(*####################### Folgende Werte sind Regelparameter und müssen initialisiert werden##########################*)
	T_ZYKL: REAL:=0.001;(*Zykluszeit in s, in der dieser Baustein aufgerufen wird*)
	C_INVERS:BOOL:=FALSE; (*Zählrichtungsumkehr*)
	IBW:LREAL:=0.1; (*Istbewertung in mm pro Increment*)
	REFVEL1:REAL:=10; (*Referenzfahrtgeschwindigkeit, um Endschalter zu suchen, positive oder negative Werte:1=langsam,2=schnell*)
	REFVEL2:REAL:=-10; (*Referenzfahrtgeschwindigkeit, um vom Endschalter weg die Nullspur zu suchen,  positive oder negative Werte:1=langsam,2=schnel*)
	REF_ON:BOOL; (*Referenzfahrt ohne Nullspur, d.h. bei negtiver Flanke des Endsch. wird Istwert gesetzt*)
	OPTI_KURZ:BOOL;(*optimierung bei kurzer Strecke:Ist der Verfahrweg kleiner als 2*S_SCHLEICH, dann wird auf halbem Weg beschleunugt(EIL) und auf halbem abgebremst (SCHLEICH*)
	WAITTIME_INV:REAL:=0.3;(*Wartezeit bei Richtungsumkehr in SEC*)
	WAIT_Restart_akt:BOOL;(* Wartezeit bei wiederStarten aktiv: wenn der Antrieb abgeschaltet wird, dann bleiben die Ausgänge MINDESTENS "Waittime_INV" abgeschaltet (notwendig bei 24V-DC Lineramotoren) *)
	S_SCHLEICH: REAL;(*Schleichweg*)
	S_STOP: REAL;(*Vorabschaltdifferenz, innerhalb diesem Fenster wird nicht positioniert, sondern PEH ausgegeben!*)
	T_VERZ_STILL:REAL;(*Verzögerungszeit zum Ansprechen der Stillstandsüberwachung, Sekunden*)
	IstWertOffset:LREAL;(*Offset, der  auf den Istwert(Benutzereinheit bzw. mm) Online aufgerechnent wird*)
	MaxIstDiff_pro_Zykl: REAL;(*Einheit: Benutzer (mm) . Wenn zwischen 2 Zyklen eine Istwertänderung (Benutzereinheit bzw. mm) von mehr als dieser Wert auftritt, wird SYNC gelöscht*)
	Loop_val: REAL;		(*schleife fahren: 0=nein; ansonsten: Es wird um den Betrag von S_STOP+Loop_Val vom Ziel weggefahren, abhängig vom Vorzeiche: + in pos.
							Richtung,- in neg. Richtung). Loop_val wird nur bei pos. Flanke Start oder Änderung der Sollpos bei aktivem Start ausgewertet, d.h. eine Änderung während dem Positionieren wird ignoriert*)
END_VAR
VAR_OUTPUT
	DAT_TO_PLC:TES_Achse_IN;(*Übergabe der Parameter zum Anwenderprogramm *)
	COUNT_CTRL: BYTE;(*Verknüpfung mit COUNTER CTRL*)
	EIL_OUT:BOOL;(*Verknüpfung mit Ausgang schnell*)
	VOR_OUT:BOOL;(*Verknüpfung mit Ausgang vor*)
	ZUR_OUT:BOOL;(*Verknüpfung mit Ausgang zur*)
	ERR_INIT:BOOL:=TRUE;(*Fehler bei initialisierung oder noch nicht initialisiert*)
END_VAR

VAR

(*########################################Ausgangsvariabeln vom Baustein -> STRUKTUR(IN) ###################################*)
	IstPos: LREAL;(*Istposition Achse *)
	SYNC: BOOL := FALSE;
	PEH:BOOL;

(*####################################Folgende Daten werden intern berechnet und verwendet#####################################*)
	OFFSET_INC: LREAL;
	COUNT_INC: DWORD;(*Zähler-INCREMENTE*)
	COUNT_INC_LAST: DWORD;(*Zähler-INCREMENTE des letzten Zyklus, sofern Zähler-Val gültig war*)
	REFSTATUS: INT; (*0=aus,1=suche Endsch;2=Suche neg.Flanke Endsch;3=suche Nullspur,...7=beendet*)
	LAST_COUNT_CTRL: BYTE;
	V_SOLL:REAL;(*Sollgeschwindifkeit, die aufgrund der berechnungen resultiert.V_F_T wird durch V_Soll UND den zulässigen Rampen (zulässige Geschw.-Änderung pro Zyklus) berechnet*)
	Zieldiff_Pos: LREAL;(*POS-Modus: Differenz zum Ziel*)
	Start_Pos_LAST: BOOL;
	SollPos: LREAL;(*Zielposition bei Positionierung*)
	MODULOVAL_INC:REAL;(*Wert in Incrementen für MODULO-Funktion*)
	TIME_VOR: REAL;
	TIME_ZUR: REAL;
	MODULO_ERG: LREAL;
	StartFRG_Pos: BOOL;
	S_SCHLEICH_I: REAL;(*Schleichweg, Intern. Der Wert S_SCHLEICH (VAR_INPUT) wird auf S_SCHLEICH_I kopiert, außer bei optimierung für kurze Strecken *)
	T_STILLST: REAL;(* abgelaufene Stillstandszeit*)
	SetIstPos: BOOL;
	IstPos_LAST: LREAL;
	IstWertOffset_LAST: LREAL;
	Loop_akt: BOOL;(*Schleife-fahren ist aktiv*)
	c_Loop_val: REAL;(* Kopie von LoopVAL*)
	EncBitMask: DWORD;
	CountLimit1: DWORD;
	CountLimit2: DWORD;
	EmptyBits: INT;
END_VAR

SetIstPos:=FALSE;
(*Kontrolle der Parameter*)
IF T_ZYKL<=0 OR IBW<=0 THEN
	ERR_INIT:=TRUE;VOR_OUT:=FALSE;ZUR_OUT:=FALSE;EIL_OUT:=FALSE;RETURN;(*Regelparameter ungültig,Ausgänge abschalten*)
ELSE ERR_INIT:=FALSE;
END_IF
(*###################### ENDE INIT #####################################################*)

DAT_TO_PLC.STILL:=FALSE;(*Stillstand mit FALSE init.*)


EmptyBits:=(32-counter_bits);
EncBitMask:=SHR(16#FFFF_FFFF,EmptyBits); (*Bitmaske aller verwendeten Encoder-Bits *)
CountLimit1:=EncBitMask/4;(* wird für Counter-Überschlagsberechnung benutzt*)
CountLimit2:=CountLimit1*3;(* wird für Counter-Überschlagsberechnung benutzt*)

(*Zähler auswerten und konvertieren nach INC_IN, wenn RC gesetzt ist: *)
IF C_INVERS THEN 
	COUNT_INC:=DINT_TO_DWORD(-COUNT_VAL) AND EncBitMask;
ELSE 
	COUNT_INC:=DINT_TO_DWORD(COUNT_VAL)  AND EncBitMask;
END_IF
(* Überschläge zählen *)
IF COUNT_INC< CountLimit1 AND COUNT_INC_LAST>CountLimit2 THEN OFFSET_INC:=OFFSET_INC+DWORD_TO_LREAL(EncBitMask)+1.0;(*Überschlag; zum Offset einen COUNTER-Überschlagsbetrag addieren*)
ELSIF COUNT_INC>CountLimit2 AND COUNT_INC_LAST<CountLimit1 THEN OFFSET_INC:=OFFSET_INC-DWORD_TO_LREAL(EncBitMask)-1.0;(*Überschlag; vom Offset einen COUNTER-Überschlagsbetrag subtrahieren*)
END_IF

(*Stillstandsüberwachung*)
IF (VOR_OUT AND (COUNT_INC<=COUNT_INC_LAST)) OR (ZUR_OUT AND (COUNT_INC>=COUNT_INC_LAST)) THEN
	T_STILLST:=T_STILLST + T_ZYKL;
	DAT_TO_PLC.STILL:=T_STILLST>T_VERZ_STILL; (*Stillstandsüberwachungszeit abgelaufen ?->SET Stillstand*)
ELSE
	T_STILLST:=0;
END_IF
LAST_COUNT_CTRL:=COUNT_CTRL;

(*############# Referenzmodus: ohne Nullspur oder mit Nullspur ( mit EL,LV COUNTER) #############*)
IF DAT_FROM_PLC.REF THEN
	IF NOT REF_ON THEN (*Referenz mit Nullspur*)
		IF REFSTATUS=0 THEN (*Referenzfahrt hat noch nicht begonnen*)
			SYNC:=FALSE;(*Sync löschen bei Anwahl von Ref-Modus*)
			IF NOT EREF THEN REFSTATUS:=1; (*Refstatus: suche Endschalter*)
			ELSE REFSTATUS:=2; (*Refstatus: Endschalter belegt, suche negative Flanke Endschalter*)
			END_IF
		ELSIF REFSTATUS=1 AND EREF THEN REFSTATUS:=2; (*Wenn Status=suche Endschalter und EREF belegt, dann Status=2*)
		ELSIF REFSTATUS=2 AND NOT EREF THEN REFSTATUS:=3;COUNT_CTRL:=0; (*negative Flanke Endschalter: Nullspur suchen, Status=3, EL  löschen und warten bis L_VALID=0 wird*)
		ELSIF REFSTATUS=3 AND (COUNT_STATE AND 1) = 0 THEN COUNT_CTRL:=1;REFSTATUS:=4;(*LV ist 0, d.h. EL=FALSE wurde angenommen, jetzt muß EL gesetzt werden, damit bei nächster Nullspur LV=1 wird!!!*)
		ELSIF REFSTATUS=4 AND (COUNT_STATE AND 1) <> 0 THEN REFSTATUS:=6; (*LV wurde gültig, jetzt kann  LATCH gelesen werden*)
			(*Offset durch LATCH-Wert neu berechnen*)
			IF C_INVERS THEN OFFSET_INC:=(DAT_FROM_PLC.Refpos/IBW)-(16#FFFF-COUNT_LATCH);COUNT_INC:=16#00FFFF-COUNT_LATCH;
			ELSE OFFSET_INC:=(DAT_FROM_PLC.Refpos/IBW)-COUNT_LATCH;COUNT_INC:=COUNT_LATCH;END_IF
			REFSTATUS:=7;SYNC:=TRUE;SetIstPos:=TRUE;
		END_IF
	ELSE (*Referenz ohne Nullspur*)
		IF REFSTATUS=0 THEN (*Referenzfahrt hat noch nicht begonnen*)
			SYNC:=FALSE;(*Sync löschen bei Anwahl von Ref-Modus*)
			IF NOT EREF THEN REFSTATUS:=1; (*Refstatus: suche Endschalter*)
			ELSE REFSTATUS:=2; (*Refstatus: Endschalter belegt, suche negative Flanke Endschalter*)
			END_IF
		ELSIF REFSTATUS=1 AND EREF THEN REFSTATUS:=2; (*Wenn Status=suche Endschalter und EREF belegt, dann Status=2*)
		ELSIF REFSTATUS=2 AND NOT EREF THEN
			 REFSTATUS:=7; (*negative Flanke Endschalter: Refstatus=7 (fertig, Istwert neu setzen*)
			OFFSET_INC:=DAT_FROM_PLC.RefPos/IBW-COUNT_INC;SYNC:=TRUE;SetIstPos:=TRUE;
		END_IF
	END_IF
ELSE REFSTATUS:=0;COUNT_CTRL:=0; (*Wenn nicht REF-Modus, dann  REFSTATUS=0*)
END_IF
(*MODULOWERT setzen*)
IF DAT_FROM_PLC.MODULO THEN
	IF ABS(COUNT_INC+OFFSET_INC)<16#7FFFFFFF THEN (*MODULO nur möglich, wenn DINT noch nicht erreicht ist*)
		MODULOVAL_INC:=MAX(DAT_FROM_PLC.MODULOVAL_INC,1);(*Div by ZERO!!!*)
		MODULO_ERG:=(LREAL_TO_DINT(COUNT_INC+OFFSET_INC))MOD REAL_TO_DINT (MODULOVAL_INC); (*Modulowert=neuer IstWert*)
		IF MODULO_ERG<0 THEN MODULO_ERG:=MODULO_ERG+MODULOVAL_INC;END_IF
		OFFSET_INC:=MODULO_ERG-COUNT_INC;SetIstPos:=TRUE;(*Offset durch den aktuellen Zählerwert neu berechnen*)
	END_IF

(*Istposition setzen*)
ELSIF DAT_FROM_PLC.SETPOS THEN
	OFFSET_INC:=DAT_FROM_PLC.RefPos/IBW-COUNT_INC;SetIstPos:=TRUE;Sync:=TRUE;
END_IF

(* Ermittlung des Geberistwertes *)
IstPos:=(COUNT_INC+OFFSET_INC)*IBW+IstWertOffset;

IF NOT SetIstPos AND (IstWertOffset=IstWertOffset_LAST) AND ABS(IstPos-IstPos_LAST) > MaxIstDiff_pro_Zykl THEN SYNC:=FALSE;END_IF

(*############################## Achsen-Steuerung ##############################################################*)
PEH:=FALSE; (*PEH mit FALSE initialisieren*)

(*################################ REFERENZFAHRT ################################################*)
IF DAT_FROM_PLC.REF AND NOT SYNC THEN
	IF REFSTATUS=1 THEN V_SOLL:=REFVEL1;
	ELSIF REFSTATUS=7 THEN V_SOLL:=0;
	ELSE V_SOLL:=REFVEL2;
	END_IF

(*########################## Positionieren auf Sollposition######################################*)
(*POSITIONIEREN POSITIONIEREN POSITIONIEREN POSITIONIEREN POSITIONIEREN POSITIONIEREN POSITIONIEREN POSITIONIEREN *)
ELSIF DAT_FROM_PLC.Start_Pos THEN
	Zieldiff_Pos:=DAT_FROM_PLC.Sollpos-IstPos;(*Reelle momentane Differenz zum Ziel*)
	IF NOT Start_Pos_LAST OR Sollpos<>DAT_FROM_PLC.Sollpos THEN (*Flanke Start oder änderung der Sollposition: Werte übergeben*)
		c_Loop_val:=Loop_val; (*Loop-Val speichern, wird während dem Positionieren ignoriert*)
		Loop_akt:=ABS(c_Loop_val) <>0 AND ABS(Zieldiff_Pos)<(S_STOP+ABS(c_Loop_val));
		SollPos:=DAT_FROM_PLC.Sollpos;DAT_TO_PLC.RET_SollPos:=Sollpos;StartFRG_Pos:=TRUE;(*Setzen der Startfreigabe*)
		IF OPTI_KURZ AND ABS(Zieldiff_Pos)<(2*S_SCHLEICH) THEN S_SCHLEICH_I:=LREAL_TO_REAL(ABS(Zieldiff_Pos)/2)+S_STOP;
		ELSE S_SCHLEICH_I:=S_SCHLEICH;
		END_IF
	END_IF

	IF ABS(Zieldiff_Pos)>(S_STOP+ABS(c_Loop_val)) THEN
		Loop_akt:=FALSE;
	END_IF

	IF Loop_akt THEN
		IF StartFRG_Pos THEN
			IF c_Loop_val > 0 THEN (*vorwärts schleife fahren*)
				V_SOLL:=1; (*langsam vor*)
			ELSE (*rückwärts schleife fahren*)
				V_SOLL:=-1; (*langsam zur*)
			END_IF
		ELSE
			V_SOLL:=0; (*keine Startfreigabe (Positionierung bereits ausgeführt), also STOP*)
		END_IF

	ELSIF ABS(Zieldiff_Pos)>S_STOP THEN (*Positionieren, STOP-Fenster noch nicht erreicht*)
		IF StartFRG_Pos THEN
			IF Zieldiff_Pos > 0 THEN (*vorwärts positionieren*)
				IF Zieldiff_Pos > S_SCHLEICH_I AND DAT_FROM_PLC.V_Pos>1 THEN V_SOLL:=2; (*schnell vor*)
				ELSE V_SOLL:=1; (*langsam vor*)
				END_IF
			ELSE (*rückwärts positionieren*)
				IF -Zieldiff_Pos > S_SCHLEICH_I AND DAT_FROM_PLC.V_Pos>1 THEN V_SOLL:=-2; (*schnell zurück*)
				ELSE V_SOLL:=-1; (*langsam zurück*)
				END_IF
			END_IF
		ELSE
			V_SOLL:=0; (*keine Startfreigabe (Positionierung bereits ausgeführt), also STOP*)
		END_IF
	ELSE  (*S_STOP-Fenster bereits erreicht*)
		PEH:=TRUE;
		V_SOLL:=0;
		StartFRG_Pos:=FALSE;
	END_IF


(*################### JOG-Betrieb mit konstanter Geschwindigkeit ohne Startrampe ###################*)
(* JOG JOG JOG JOG JOG JOG JOG JOG JOG JOG JOG JOG JOG JOG JOG JOG JOG JOG JOG JOG JOG JOG JOG JOG JOG JOG JOG *)
ELSIF DAT_FROM_PLC.JOGFW THEN
	V_SOLL:=DAT_FROM_PLC.V_JOG;

ELSIF DAT_FROM_PLC.JOGBW THEN
	V_SOLL:=-DAT_FROM_PLC.V_JOG;

(*####################### Anhalten, keine Bedingung erfüllt##########################################*)
(* HALT HALT HALT HALT HALT HALT HALT HALT HALT HALT HALT HALT HALT HALT HALT HALT HALT HALT HALT HALT HALT HALT *)
ELSE V_SOLL:=0;
END_IF


(*########## Berechnung der Ausgänge ###############*)
IF V_SOLL > 0 THEN (*Sollgeschwindigkeit vor*)
	IF TIME_ZUR=0 AND (TIME_VOR=0 OR  NOT WAIT_Restart_akt OR VOR_OUT) THEN (*keine Richtungsumkehr, rückwärts-Wartezeit ist abgelaufen UND keine wartezeit Restart oder abgelaufen oder fährt bereits*)
		(*positionieren vor*)
		TIME_VOR:=WAITTIME_INV;(*Wartezeit laden*)
		IF V_SOLL=2 THEN DAT_TO_PLC.VEL_IST:=2;
		ELSE DAT_TO_PLC.VEL_IST:=1;
		END_IF
	ELSE (*Rückwärts-Wartezeit läuft noch*)
		DAT_TO_PLC.VEL_IST:=0;
	END_IF
ELSIF V_SOLL < 0 THEN(*Sollgeschwindigkeit negativ*)
	IF TIME_VOR=0 AND (TIME_ZUR=0 OR  NOT WAIT_Restart_akt OR ZUR_OUT) THEN (*keine Richtungsumkehr, vorwärts-Wartezeit ist abgelaufen UND keine wartezeit Restart oder abgelaufen oder fährt bereits*)
		(*positionieren zurück*)
		TIME_ZUR:=WAITTIME_INV;(*Wartezeit "zurück" laden*)
		IF V_SOLL=-2 THEN DAT_TO_PLC.VEL_IST:=-2;
		ELSE DAT_TO_PLC.VEL_IST:=-1;
		END_IF
	ELSE (*vorwärts-Wartezeit läuft noch*)
		DAT_TO_PLC.VEL_IST:=0;
	END_IF
ELSE (*Sollgeschwindigkeit = 0, also STOP*)
	DAT_TO_PLC.VEL_IST:=0;
END_IF
(*Wartezeit decrementieren*)
TIME_VOR:=MAX((TIME_VOR-T_ZYKL),0);TIME_ZUR:=MAX((TIME_ZUR-T_ZYKL),0);
(*Zyklusverz. Var.*)
COUNT_INC_LAST:=COUNT_INC;
Start_Pos_LAST:=DAT_FROM_PLC.Start_Pos;

(*Ausgangsvariablen übergeben*)
DAT_TO_PLC.IstPos:=IstPos;
DAT_TO_PLC.SYNC:=SYNC;
DAT_TO_PLC.PEH:=PEH;
(*Ausgänge setzen*)
VOR_OUT:=DAT_TO_PLC.VEL_IST>0;
ZUR_OUT:=DAT_TO_PLC.VEL_IST<0;
EIL_OUT:=ABS(DAT_TO_PLC.VEL_IST)>=2;
IstPos_Last:=IstPos;
IstWertOffset_LAST:=IstWertOffset;

END_FUNCTION_BLOCK

// POUs/Achsen_Bausteinen/ES_KL2552
FUNCTION_BLOCK ES_KL2552 (*Eil-Schleich - Achse für DC-Klemme 2552. CTRL wird nur gelesen, Baustein wird nicht bearbeitet wenn Registecom aktiv ist.*)
VAR_INPUT
	DAT_FROM_PLC:TES_Achse_OUT; (*Übergabe der Parameter vom Anwenderprogramm *)
	COUNT_VAL: DINT;(*Verknüpfung mit COUNTER VAL*)
	COUNT_STATE: BYTE;(*Verknüpfung mit COUNTER STATE*)
	COUNT_CTRL: BYTE;(*Verknüpfung mit COUNTER CTRL*)
	EREF: BOOL; (*Verknüpfung mit Referenzeingang*)

(*####################### Folgende Werte sind Regelparameter und müssen initialisiert werden##########################*)
	T_ZYKL: REAL:=0.001;(*Zykluszeit in s, in der dieser Baustein aufgerufen wird*)
	C_INVERS:BOOL:=FALSE; (*Zählrichtungsumkehr*)
	IBW:LREAL:=0.1; (*Istbewertung in mm pro Increment*)
	REFVEL1:REAL:=10; (*Referenzfahrtgeschwindigkeit, um Endschalter zu suchen, positive oder negative Werte:1=langsam,2=schnell*)
	REFVEL2:REAL:=-10; (*Referenzfahrtgeschwindigkeit, um vom Endschalter weg die Nullspur zu suchen,  positive oder negative Werte:1=langsam,2=schnel*)
	OPTI_KURZ:BOOL;(*optimierung bei kurzer Strecke:Ist der Verfahrweg kleiner als 2*S_SCHLEICH, dann wird auf halbem Weg beschleunugt(EIL) und auf halbem abgebremst (SCHLEICH*)
	WAITTIME_INV:REAL:=0.3;(*Wartezeit bei Richtungsumkehr in SEC*)
	S_SCHLEICH: REAL;(*Schleichweg*)
	S_STOP: REAL;(*Vorabschaltdifferenz, innerhalb diesem Fenster wird nicht positioniert, sondern PEH ausgegeben!*)
	T_VERZ_STILL:REAL;(*Verzögerungszeit zum Ansprechen der Stillstandsüberwachung, Sekunden*)
	IstWertOffset:LREAL;(*Offset, der  auf den Istwert(Benutzereinheit bzw. mm) Online aufgerechnent wird*)
	MaxIstDiff_pro_Zykl: REAL;(*Einheit: Benutzer (mm).Wenn zwischen 2 Zyklen eine Istwertänderung (Benutzereinheit bzw. mm) von mehr als dieser Wert auftritt, wird SYNC gelöscht*)
	nSoll_Invers:BOOL;
	ACC: REAL;		(*Beschleunigung/Verzögerung: in %/sec*)
END_VAR
VAR_OUTPUT
	DAT_TO_PLC:TES_Achse_IN;(*Übergabe der Parameter zum Anwenderprogramm *)
	ERR_INIT:BOOL:=TRUE;(*Fehler bei initialisierung oder noch nicht initialisiert*)
END_VAR

VAR

(*########################################Ausgangsvariabeln vom Baustein -> STRUKTUR(IN) ###################################*)
	IstPos: LREAL;(*Istposition Achse *)
	SYNC: BOOL := FALSE;
	PEH:BOOL;

(*####################################Folgende Daten werden intern berechnet und verwendet#####################################*)
	OFFSET_INC: LREAL;
	COUNT_INC: DINT;(*Zähler-INCREMENTE*)
	COUNT_INC_LAST: DINT;(*Zähler-INCREMENTE des letzten Zyklus, sofern Zähler-Val gültig war*)
	REFSTATUS: INT; (*0=aus,1=suche Endsch;2=Suche neg.Flanke Endsch;3=suche Nullspur,...7=beendet*)
	V_SOLL:REAL;(*Sollgeschwindifkeit, die aufgrund der berechnungen resultiert.V_F_T wird durch V_Soll UND den zulässigen Rampen (zulässige Geschw.-Änderung pro Zyklus) berechnet*)
	Zieldiff_Pos: LREAL;(*POS-Modus: Differenz zum Ziel*)
	Start_Pos_LAST: BOOL;
	SollPos: LREAL;(*Zielposition bei Positionierung*)
	MODULOVAL_INC:REAL;(*Wert in Incrementen für MODULO-Funktion*)
	TIME_VOR: REAL;
	TIME_ZUR: REAL;
	MODULO_ERG: LREAL;
	StartFRG_Pos: BOOL;
	S_SCHLEICH_I: REAL;(*Schleichweg, Intern. Der Wert S_SCHLEICH (VAR_INPUT) wird auf S_SCHLEICH_I kopiert, außer bei optimierung für kurze Strecken *)
	T_STILLST: REAL;(* abgelaufene Stillstandszeit*)
	SetIstPos: BOOL;
	IstPos_LAST: LREAL;
	IstWertOffset_LAST: LREAL;
END_VAR

VAR_IN_OUT
	nSoll: INT;
END_VAR

SetIstPos:=FALSE;
(*Kontrolle der Parameter*)
IF T_ZYKL<=0 OR IBW<=0 THEN
	ERR_INIT:=TRUE;nSoll:=0;RETURN;(*Regelparameter ungültig,Ausgänge abschalten*)
ELSE ERR_INIT:=FALSE;
END_IF
(*###################### ENDE INIT #####################################################*)

IF COUNT_STATE.7 OR COUNT_CTRL.7 THEN RETURN; END_IF (*Beende Baustein, da RegisterKommunikation aktiv ist. *)

DAT_TO_PLC.STILL:=FALSE;(*Stillstand mit FALSE init.*)


(*Zähler auswerten und konvertieren nach INC_IN, wenn RC gesetzt ist: *)
IF C_INVERS THEN COUNT_INC:=16#FFFF-COUNT_VAL;ELSE COUNT_INC:=COUNT_VAL;END_IF
(* Überschläge zählen *)
IF COUNT_INC< 16000 AND COUNT_INC_LAST>48000 THEN OFFSET_INC:=OFFSET_INC+16#10000;(*Überschlag; zum Offset einen COUNTER-Überschlagsbetrag addieren*)
ELSIF COUNT_INC>48000 AND COUNT_INC_LAST<16000 THEN OFFSET_INC:=OFFSET_INC-16#10000;(*Überschlag; vom Offset einen COUNTER-Überschlagsbetrag subtrahieren*)
END_IF



(*Stillstandsüberwachung*)
IF ((DAT_TO_PLC.VEL_IST > 0 ) AND (COUNT_INC<=COUNT_INC_LAST)) OR ((DAT_TO_PLC.VEL_IST < 0) AND (COUNT_INC>=COUNT_INC_LAST)) THEN
	T_STILLST:=T_STILLST + T_ZYKL;
	DAT_TO_PLC.STILL:=T_STILLST>T_VERZ_STILL; (*Stillstandsüberwachungszeit abgelaufen ?->SET Stillstand*)
ELSE
	T_STILLST:=0;
END_IF


(*############# Referenzmodus: ohne Nullspur oder mit Nullspur ( mit EL,LV COUNTER) #############*)
IF DAT_FROM_PLC.REF THEN
 (*Referenz ohne Nullspur*)
	IF REFSTATUS=0 THEN (*Referenzfahrt hat noch nicht begonnen*)
		SYNC:=FALSE;(*Sync löschen bei Anwahl von Ref-Modus*)
		IF NOT EREF THEN REFSTATUS:=1; (*Refstatus: suche Endschalter*)
		ELSE REFSTATUS:=2; (*Refstatus: Endschalter belegt, suche negative Flanke Endschalter*)
		END_IF
	ELSIF REFSTATUS=1 AND EREF THEN REFSTATUS:=2; (*Wenn Status=suche Endschalter und EREF belegt, dann Status=2*)
	ELSIF REFSTATUS=2 AND NOT EREF THEN
		 REFSTATUS:=7; (*negative Flanke Endschalter: Refstatus=7 (fertig, Istwert neu setzen*)
		OFFSET_INC:=DAT_FROM_PLC.RefPos/IBW-COUNT_INC;SYNC:=TRUE;SetIstPos:=TRUE;
	END_IF
ELSE REFSTATUS:=0; (*Wenn nicht REF-Modus, dann  REFSTATUS=0*)
END_IF
(*MODULOWERT setzen*)
IF DAT_FROM_PLC.MODULO THEN
	IF ABS(COUNT_INC+OFFSET_INC)<16#7FFFFFFF THEN (*MODULO nur möglich, wenn DINT noch nicht erreicht ist*)
		MODULOVAL_INC:=MAX(DAT_FROM_PLC.MODULOVAL_INC,1);(*Div by ZERO!!!*)
		MODULO_ERG:=(LREAL_TO_DINT(COUNT_INC+OFFSET_INC))MOD REAL_TO_DINT (MODULOVAL_INC); (*Modulowert=neuer IstWert*)
		IF MODULO_ERG<0 THEN MODULO_ERG:=MODULO_ERG+MODULOVAL_INC;END_IF
		OFFSET_INC:=MODULO_ERG-COUNT_INC;SetIstPos:=TRUE;(*Offset durch den aktuellen Zählerwert neu berechnen*)
	END_IF

(*Istposition setzen*)
ELSIF DAT_FROM_PLC.SETPOS THEN
	OFFSET_INC:=DAT_FROM_PLC.RefPos/IBW-COUNT_INC;SetIstPos:=TRUE;Sync:=TRUE;
END_IF

(* Ermittlung des Geberistwertes *)
IstPos:=(COUNT_INC+OFFSET_INC)*IBW+IstWertOffset;

IF NOT SetIstPos AND (IstWertOffset=IstWertOffset_LAST) AND ABS(IstPos-IstPos_LAST) > MaxIstDiff_pro_Zykl THEN SYNC:=FALSE;END_IF


(*############################## Achsen-Steuerung ##############################################################*)
PEH:=FALSE; (*PEH mit FALSE initialisieren*)

(*################################ REFERENZFAHRT ################################################*)
IF DAT_FROM_PLC.REF AND NOT SYNC THEN
	IF REFSTATUS=1 THEN V_SOLL:=REFVEL1;
	ELSIF REFSTATUS=7 THEN V_SOLL:=0;
	ELSE V_SOLL:=REFVEL2;
	END_IF














(*########################## Positionieren auf Sollposition######################################*)
(*POSITIONIEREN POSITIONIEREN POSITIONIEREN POSITIONIEREN POSITIONIEREN POSITIONIEREN POSITIONIEREN POSITIONIEREN *)
ELSIF DAT_FROM_PLC.Start_Pos THEN
	Zieldiff_Pos:=DAT_FROM_PLC.Sollpos-IstPos;(*Reelle momentane Differenz zum Ziel*)
	IF NOT Start_Pos_LAST OR Sollpos<>DAT_FROM_PLC.Sollpos THEN (*Flanke Start oder änderung der Sollposition: Werte übergeben*)
		SollPos:=DAT_FROM_PLC.Sollpos;DAT_TO_PLC.RET_SollPos:=Sollpos;StartFRG_Pos:=TRUE;(*Setzen der Startfreigabe*)
		IF OPTI_KURZ AND ABS(Zieldiff_Pos)<(2*S_SCHLEICH) THEN S_SCHLEICH_I:=LREAL_TO_REAL(ABS(Zieldiff_Pos)/2)+S_STOP;
		ELSE S_SCHLEICH_I:=S_SCHLEICH;
		END_IF
	END_IF
	IF ABS(Zieldiff_Pos)>S_STOP THEN (*Positionieren, STOP-Fenster noch nicht erreicht*)
		IF StartFRG_Pos THEN
			IF Zieldiff_Pos > 0 THEN (*vorwärts positionieren*)
				IF Zieldiff_Pos > S_SCHLEICH_I THEN V_SOLL:=DAT_FROM_PLC.V_Pos; (*schnell vor*)
				ELSE V_SOLL:=DAT_FROM_PLC.V_JOG; (*langsam vor*)
				END_IF
			ELSE (*rückwärts positionieren*)
				IF -Zieldiff_Pos > S_SCHLEICH_I THEN V_SOLL:=-DAT_FROM_PLC.V_Pos; (*schnell zurück*)
				ELSE V_SOLL:=-DAT_FROM_PLC.V_JOG; (*langsam zurück*)
				END_IF
			END_IF
		ELSE
			V_SOLL:=0; (*keine Startfreigabe (Positionierung bereits ausgeführt), also STOP*)
		END_IF
	ELSE  (*S_STOP-Fenster bereits erreicht*)
		PEH:=TRUE;
		V_SOLL:=0;
		StartFRG_Pos:=FALSE;
	END_IF


(*################### JOG-Betrieb mit konstanter Geschwindigkeit ohne Startrampe ###################*)
(* JOG JOG JOG JOG JOG JOG JOG JOG JOG JOG JOG JOG JOG JOG JOG JOG JOG JOG JOG JOG JOG JOG JOG JOG JOG JOG JOG *)
ELSIF DAT_FROM_PLC.JOGFW THEN
	V_SOLL:=DAT_FROM_PLC.V_JOG;

ELSIF DAT_FROM_PLC.JOGBW THEN
	V_SOLL:=-DAT_FROM_PLC.V_JOG;

(*####################### Anhalten, keine Bedingung erfüllt##########################################*)
(* HALT HALT HALT HALT HALT HALT HALT HALT HALT HALT HALT HALT HALT HALT HALT HALT HALT HALT HALT HALT HALT HALT *)
ELSE V_SOLL:=0;
END_IF


(*########## Berechnung der Ausgänge ###############*)
IF V_SOLL > 0 THEN (*Sollgeschwindigkeit vor*)
	IF TIME_ZUR=0 THEN (*keine Richtungsumkehr, rückwärts-Wartezeit ist abgelaufen*)
		(*positionieren vor*)
		TIME_VOR:=WAITTIME_INV;(*Wartezeit laden*)
		DAT_TO_PLC.VEL_IST:=LREAL_TO_REAL(LIMIT((DAT_TO_PLC.VEL_IST-T_ZYKL*ACC),V_SOLL,(DAT_TO_PLC.VEL_IST+T_ZYKL*ACC)));
	ELSE (*Rückwärts-Wartezeit läuft noch*)
		DAT_TO_PLC.VEL_IST:=LREAL_TO_REAL(LIMIT((DAT_TO_PLC.VEL_IST-T_ZYKL*ACC),0.0,(DAT_TO_PLC.VEL_IST+T_ZYKL*ACC)));
	END_IF
ELSIF V_SOLL < 0 THEN(*Sollgeschwindigkeit negativ*)
	IF TIME_VOR=0 THEN (*keine Richtungsumkehr, vorwärts-Wartezeit ist abgelaufen*)
		(*positionieren zurück*)
		TIME_ZUR:=WAITTIME_INV;(*Wartezeit "zurück" laden*)
		DAT_TO_PLC.VEL_IST:=LREAL_TO_REAL(LIMIT((DAT_TO_PLC.VEL_IST-T_ZYKL*ACC),V_SOLL,(DAT_TO_PLC.VEL_IST+T_ZYKL*ACC)));
	ELSE (*vorwärts-Wartezeit läuft noch*)
		DAT_TO_PLC.VEL_IST:=LREAL_TO_REAL(LIMIT((DAT_TO_PLC.VEL_IST-T_ZYKL*ACC),0.0,(DAT_TO_PLC.VEL_IST+T_ZYKL*ACC)));
	END_IF
ELSE (*Sollgeschwindigkeit = 0, also STOP*)
		DAT_TO_PLC.VEL_IST:=LREAL_TO_REAL(LIMIT((DAT_TO_PLC.VEL_IST-T_ZYKL*ACC),0.0,(DAT_TO_PLC.VEL_IST+T_ZYKL*ACC)));
END_IF
(*Wartezeit decrementieren*)
TIME_VOR:=MAX((TIME_VOR-T_ZYKL),0);TIME_ZUR:=MAX((TIME_ZUR-T_ZYKL),0);
(*Zyklusverz. Var.*)
COUNT_INC_LAST:=COUNT_INC;
Start_Pos_LAST:=DAT_FROM_PLC.Start_Pos;

(*Ausgangsvariablen übergeben*)
DAT_TO_PLC.IstPos:=IstPos;
DAT_TO_PLC.SYNC:=SYNC;
DAT_TO_PLC.PEH:=PEH;
(*Ausgänge setzen*)

nSoll:=REAL_TO_INT(LIMIT(-32767.0,(DAT_TO_PLC.VEL_IST*327.67),32767.0));
IF nSoll_Invers THEN nSoll:=-nSoll; END_IF
IstPos_Last:=IstPos;

IstWertOffset_LAST:=IstWertOffset;

END_FUNCTION_BLOCK

// POUs/Achsen_Bausteinen/ES_KL5001_A
FUNCTION_BLOCK ES_KL5001_A(*Eil-Schleich - Achse für KL5001*)
VAR_INPUT
	DAT_FROM_PLC:TES_Achse_OUT; (*Übergabe der Parameter vom Anwenderprogramm *)
	VAL_HI: WORD;(*Verknüpfung mit VAL HI*)
	VAL_LO: WORD;(*Verknüpfung mit VAL LO*)

(*####################### Folgende Werte sind Regelparameter und müssen initialisiert werden##########################*)
	T_ZYKL: REAL:=0.001;(*Zykluszeit in s, in der dieser Baustein aufgerufen wird*)
	C_INVERS:BOOL:=FALSE; (*Zählrichtungsumkehr*)
	IBW:LREAL:=0.1; (*Istbewertung in mm pro Increment*)
	OPTI_KURZ:BOOL;(*optimierung bei kurzer Strecke:Ist der Verfahrweg kleiner als 2*S_SCHLEICH, dann wird auf halbem Weg beschleunugt(EIL) und auf halbem abgebremst (SCHLEICH*)
	WAITTIME_INV:REAL:=0.3;(*Wartezeit bei Richtungsumkehr in SEC*)
	S_SCHLEICH: REAL;(*Schleichweg*)
	S_STOP: REAL;(*Vorabschaltdifferenz, innerhalb diesem Fenster wird nicht positioniert, sondern PEH ausgegeben!*)
	T_VERZ_STILL:REAL;(*Verzögerungszeit zum Ansprechen der Stillstandsüberwachung, Sekunden*)
	IstWertOffset:LREAL;(*Offset, der  auf den Istwert(Benutzereinheit bzw. mm) Online aufgerechnent wird*)
	SSI_MAX_DIFF: DINT; (*Einheit: Incremente. Zur Überbrückung des SSI-Encoderfehlers bei Überschlag: Wenn Incremente-Sprung > SSI_MAX_DIFF, dann wird der Geberistwert eingefrohren bis wieder der richtige Wert gemeldet wird oder bis TIMEOUT überschritten ist*)
	MAX_FREESTIME_SMD_sec: REAL;(* "Ssi-Max-Differenz":Zur Überbrückung des SSI-Encoderfehlers bei Überschlag: Für maximal diese Zeit wird der Istwert eingefroren wenn er einen Sprung macht der grösser SSI_MAX_DIFF ist*)
	Loop_val: REAL;		(*schleife fahren: 0=nein; ansonsten: Es wird um den Betrag von S_STOP+Loop_Val vom Ziel weggefahren, abhängig vom Vorzeiche: + in pos.
							Richtung,- in neg. Richtung). Loop_val wird nur bei pos. Flanke Start oder Änderung der Sollpos bei aktivem Start ausgewertet, d.h. eine Änderung während dem Positionieren wird ignoriert*)
	IWTyp: REAL;(*Istwert Typisch: Dieser Wert ist Notwendig, um den Geberüberschlag intern ausserhalb dem typischen Istwert zu verschieben, er kann
				 mit0 (oder gar nicht = 0) parametriert werden. Nur in Sonderfällen, wo aufgrund einem hohen Verfahrweg der gesamte Geberbereich abgefahren wird, kann es notwendig sein, einen korrekten Wert anzugeben. In 
				diesem fall ist der Mittelwert zwischen Minpos und Maxpos anzugeben; eine Achse, die in diesem Fall z.B. von +20000mm bis +60000 mm verfährt, muss dann mit +40000 parametriert werden. Die maximale Anzahl der möglichen Incremente des Gebers sollte
				auf jeden Fall kontrolliert werden.*)
	Geber24Bit:BOOL;(* Es ist ein Geber angeschlossen, der nur 24-Bit liefert, d.h. der Überschlag des Gebers erfolgt nach 24 Bits: 16#00FF_FFFF -> 16#0000_0000*)
END_VAR
VAR_OUTPUT
	DAT_TO_PLC:TES_Achse_IN;(*Übergabe der Parameter zum Anwenderprogramm *)
	EIL_OUT:BOOL;(*Verknüpfung mit Ausgang schnell*)
	VOR_OUT:BOOL;(*Verknüpfung mit Ausgang vor*)
	ZUR_OUT:BOOL;(*Verknüpfung mit Ausgang zur*)
	ERR_INIT:BOOL:=TRUE;(*Fehler bei initialisierung oder noch nicht initialisiert*)
END_VAR

VAR

(*########################################Ausgangsvariabeln vom Baustein -> STRUKTUR(IN) ###################################*)
	IstPos: LREAL;(*Istposition Achse *)
	SYNC: BOOL := FALSE;
	PEH:BOOL;

(*####################################Folgende Daten werden intern berechnet und verwendet#####################################*)
	COUNT_VAL: DWORD;(*Zähler-INCREMENTE*)
	COUNT_INC: DINT;(*Zähler-INCREMENTE*)
	COUNT_INC_LAST: DINT;(*Zähler-INCREMENTE des letzten Zyklus, sofern Zähler-Val gültig war*)
	V_SOLL:REAL;(*Sollgeschwindifkeit, die aufgrund der berechnungen resultiert.V_F_T wird durch V_Soll UND den zulässigen Rampen (zulässige Geschw.-Änderung pro Zyklus) berechnet*)
	Zieldiff_Pos: LREAL;(*POS-Modus: Differenz zum Ziel*)
	Start_Pos_LAST: BOOL;
	SollPos: LREAL;(*Zielposition bei Positionierung*)
	TIME_VOR: REAL;
	TIME_ZUR: REAL;
	StartFRG_Pos: BOOL;
	S_SCHLEICH_I: REAL;(*Schleichweg, Intern. Der Wert S_SCHLEICH (VAR_INPUT) wird auf S_SCHLEICH_I kopiert, außer bei optimierung für kurze Strecken *)
	T_STILLST: REAL;(* abgelaufene Stillstandszeit*)
	SetIstPos: BOOL;
	IstPos_LAST: LREAL;
	IstWertOffset_LAST: LREAL;
	TIMECOUNT_SMD: LREAL;
	Loop_akt: BOOL;(*Schleife-fahren ist aktiv*)
	c_Loop_val: REAL;(* Kopie von LoopVAL*)
	IncOffset: DINT;
	IBW2: LREAL;
END_VAR

SetIstPos:=FALSE;
(*Kontrolle der Parameter*)
IF T_ZYKL<=0 OR IBW<=0 THEN
	ERR_INIT:=TRUE;VOR_OUT:=FALSE;ZUR_OUT:=FALSE;EIL_OUT:=FALSE;RETURN;(*Regelparameter ungültig,Ausgänge abschalten*)
ELSE ERR_INIT:=FALSE;
END_IF
(*###################### ENDE INIT #####################################################*)

DAT_TO_PLC.STILL:=FALSE;(*Stillstand mit FALSE init.*)

COUNT_VAL:=VAL_HI*16#10000+VAL_LO;(*COUNT_INC aus HI und LO-Werten errechnen*)

IF Geber24Bit THEN
	COUNT_VAL:=SHL(COUNT_VAL,8);
	IBW2:=IBW/256;
ELSE
	IBW2:=IBW;
END_IF


IncOffset:=LREAL_TO_DINT((IstWertOffset-IWTyp)/IBW2)+DWORD_TO_DINT(16#8000_0000);(*Der Istwertoffset, der Betrag der Typschen Position und die Hälfte des Gesamt-Icnremente-Bereichs müssen aufgerechnet werden, damit kein Überschlag möglich ist*)
IF C_INVERS THEN
	COUNT_INC:=DWORD_TO_DINT(16#FFFF_FFFF) - (DWORD_TO_DINT(COUNT_VAL)-IncOffset);
ELSE
	COUNT_INC:=DWORD_TO_DINT(Count_Val)+IncOffset;
END_IF

(*Stillstandsüberwachung*)
IF (VOR_OUT AND (COUNT_INC<=COUNT_INC_LAST)) OR (ZUR_OUT AND (COUNT_INC>=COUNT_INC_LAST)) THEN
	T_STILLST:=T_STILLST + T_ZYKL;
	DAT_TO_PLC.STILL:=T_STILLST>T_VERZ_STILL; (*Stillstandsüberwachungszeit abgelaufen ?->SET Stillstand*)
ELSE
	T_STILLST:=0;
END_IF

IF ABS (COUNT_INC-COUNT_INC_LAST) > SSI_MAX_DIFF AND TIMECOUNT_SMD<MAX_FREESTIME_SMD_sec THEN
	(*Der Istwertsprung des SSI-Gebers ist > der angegebenen Differenz und die maximale Frierzeit ist noch nicht abgelaufen. Für die Angegebene Zeit wird der Istwert eingefrohren bzw. dem Sollwert nachgeführt*)
	TIMECOUNT_SMD:=TIMECOUNT_SMD+T_ZYKL; (*Zählen der laufeneden Frier-Zeit*)
ELSE (*Istwertberechnung ausführen, denn SSI_MAX_DIFF ist nicht überschritten oder MAX_FREESTIME_SMD ist abgelaufen*)
	TIMECOUNT_SMD:=0; (*Zeitzähler nullen*)
	(*Freese bei ONLINE-Istwertoffsetänderung, damit sich die Position des Antriebes nicht mechanisch verändert*)

	(* Ermittlung des Geberistwertes *)
	IstPos:=DINT_TO_LREAL(COUNT_INC-DWORD_TO_DINT(16#8000_0000))*IBW2+IWTyp;(* Der Istwertoffset ist bereits den Incrementwert aufgerechnet, der halbe Gesamtincrement-Bereich und der Typ.Istwert, die ebenfalls aufgerechnet wurden, müss hier wieder abgerechnet werden: 2147483648 D = 16#8000_0000 H*)
	IstWertOffset_LAST:=IstWertOffset;
	COUNT_INC_LAST:=COUNT_INC; (*COUNT_INC_LAST zuweisen*)
END_IF



















































(*############################## Achsen-Steuerung ##############################################################*)
PEH:=FALSE; (*PEH mit FALSE initialisieren*)

(*########################## Positionieren auf Sollposition######################################*)
(*POSITIONIEREN POSITIONIEREN POSITIONIEREN POSITIONIEREN POSITIONIEREN POSITIONIEREN POSITIONIEREN POSITIONIEREN *)
IF DAT_FROM_PLC.Start_Pos THEN
	Zieldiff_Pos:=DAT_FROM_PLC.Sollpos-IstPos;(*Reelle momentane Differenz zum Ziel*)
	IF NOT Start_Pos_LAST OR Sollpos<>DAT_FROM_PLC.Sollpos THEN (*Flanke Start oder änderung der Sollposition: Werte übergeben*)
		c_Loop_val:=Loop_val; (*Loop-Val speichern, wird während dem Positionieren ignoriert*)
		Loop_akt:=ABS(c_Loop_val) <>0 AND ABS(Zieldiff_Pos)<(S_STOP+ABS(c_Loop_val));
		SollPos:=DAT_FROM_PLC.Sollpos;DAT_TO_PLC.RET_SollPos:=Sollpos;StartFRG_Pos:=TRUE;(*Setzen der Startfreigabe*)
		IF OPTI_KURZ AND ABS(Zieldiff_Pos)<(2*S_SCHLEICH) THEN S_SCHLEICH_I:=LREAL_TO_REAL(ABS(Zieldiff_Pos)/2)+S_STOP;
		ELSE S_SCHLEICH_I:=S_SCHLEICH;
		END_IF
	END_IF

	IF ABS(Zieldiff_Pos)>(S_STOP+ABS(c_Loop_val)) THEN
		Loop_akt:=FALSE;
	END_IF

	IF Loop_akt THEN
		IF StartFRG_Pos THEN
			IF c_Loop_val > 0 THEN (*vorwärts schleife fahren*)
				V_SOLL:=1; (*langsam vor*)
			ELSE (*rückwärts schleife fahren*)
				V_SOLL:=-1; (*langsam zur*)
			END_IF
		ELSE
			V_SOLL:=0; (*keine Startfreigabe (Positionierung bereits ausgeführt), also STOP*)
		END_IF

	ELSIF ABS(Zieldiff_Pos)>S_STOP THEN (*Positionieren, STOP-Fenster noch nicht erreicht*)
		IF StartFRG_Pos THEN
			IF Zieldiff_Pos > 0 THEN (*vorwärts positionieren*)
				IF Zieldiff_Pos > S_SCHLEICH_I AND DAT_FROM_PLC.V_Pos>1 THEN V_SOLL:=2; (*schnell vor*)
				ELSE V_SOLL:=1; (*langsam vor*)
				END_IF
			ELSE (*rückwärts positionieren*)
				IF -Zieldiff_Pos > S_SCHLEICH_I AND DAT_FROM_PLC.V_Pos>1 THEN V_SOLL:=-2; (*schnell zurück*)
				ELSE V_SOLL:=-1; (*langsam zurück*)
				END_IF
			END_IF
		ELSE
			V_SOLL:=0; (*keine Startfreigabe (Positionierung bereits ausgeführt), also STOP*)
		END_IF
	ELSE  (*S_STOP-Fenster bereits erreicht*)
		PEH:=TRUE;
		V_SOLL:=0;
		StartFRG_Pos:=FALSE;
	END_IF


(*################### JOG-Betrieb mit konstanter Geschwindigkeit ohne Startrampe ###################*)
(* JOG JOG JOG JOG JOG JOG JOG JOG JOG JOG JOG JOG JOG JOG JOG JOG JOG JOG JOG JOG JOG JOG JOG JOG JOG JOG JOG *)
ELSIF DAT_FROM_PLC.JOGFW THEN
	V_SOLL:=DAT_FROM_PLC.V_JOG;

ELSIF DAT_FROM_PLC.JOGBW THEN
	V_SOLL:=-DAT_FROM_PLC.V_JOG;

(*####################### Anhalten, keine Bedingung erfüllt##########################################*)
(* HALT HALT HALT HALT HALT HALT HALT HALT HALT HALT HALT HALT HALT HALT HALT HALT HALT HALT HALT HALT HALT HALT *)
ELSE V_SOLL:=0;
END_IF


(*########## Berechnung der Ausgänge ###############*)
IF V_SOLL > 0 THEN (*Sollgeschwindigkeit vor*)
	IF TIME_ZUR=0 THEN (*keine Richtungsumkehr, rückwärts-Wartezeit ist abgelaufen*)
		(*positionieren vor*)
		TIME_VOR:=WAITTIME_INV;(*Wartezeit laden*)
		IF V_SOLL=2 THEN DAT_TO_PLC.VEL_IST:=2;
		ELSE DAT_TO_PLC.VEL_IST:=1;
		END_IF
	ELSE (*Rückwärts-Wartezeit läuft noch*)
		DAT_TO_PLC.VEL_IST:=0;
	END_IF
ELSIF V_SOLL < 0 THEN(*Sollgeschwindigkeit negativ*)
	IF TIME_VOR=0 THEN (*keine Richtungsumkehr, vorwärts-Wartezeit ist abgelaufen*)
		(*positionieren zurück*)
		TIME_ZUR:=WAITTIME_INV;(*Wartezeit "zurück" laden*)
		IF V_SOLL=-2 THEN DAT_TO_PLC.VEL_IST:=-2;
		ELSE DAT_TO_PLC.VEL_IST:=-1;
		END_IF
	ELSE (*vorwärts-Wartezeit läuft noch*)
		DAT_TO_PLC.VEL_IST:=0;
	END_IF
ELSE (*Sollgeschwindigkeit = 0, also STOP*)
	DAT_TO_PLC.VEL_IST:=0;
END_IF
(*Wartezeit decrementieren*)
TIME_VOR:=MAX((TIME_VOR-T_ZYKL),0);TIME_ZUR:=MAX((TIME_ZUR-T_ZYKL),0);
(*Zyklusverz. Var.*)

Start_Pos_LAST:=DAT_FROM_PLC.Start_Pos;

(*Ausgangsvariablen übergeben*)
DAT_TO_PLC.IstPos:=IstPos;
DAT_TO_PLC.SYNC:=SYNC;
DAT_TO_PLC.PEH:=PEH;
(*Ausgänge setzen*)
VOR_OUT:=DAT_TO_PLC.VEL_IST>0;
ZUR_OUT:=DAT_TO_PLC.VEL_IST<0;
EIL_OUT:=ABS(DAT_TO_PLC.VEL_IST)>=2;
IstPos_Last:=IstPos;

END_FUNCTION_BLOCK

// POUs/Achsen_Bausteinen/ES_KL51x1_A
FUNCTION_BLOCK ES_KL51x1_A(*Eil-Schleich - Achse für KL5101 - 5VGeber*)
VAR_INPUT
	DAT_FROM_PLC:TES_Achse_OUT; (*Übergabe der Parameter vom Anwenderprogramm *)
	COUNT_VAL: DINT;(*Verknüpfung mit COUNTER VAL*)
	COUNT_LATCH: DWORD;(*Verknüpfung mit COUNTER LATCH*)
	COUNT_STATE: BYTE;(*Verknüpfung mit COUNTER STATE*)
	EREF: BOOL; (*Verknüpfung mit Referenzeingang*)

(*####################### Folgende Werte sind Regelparameter und müssen initialisiert werden##########################*)
	T_ZYKL: REAL:=0.001;(*Zykluszeit in s, in der dieser Baustein aufgerufen wird*)
	C_INVERS:BOOL:=FALSE; (*Zählrichtungsumkehr*)
	IBW:LREAL:=0.1; (*Istbewertung in mm pro Increment*)
	REFVEL1:REAL:=10; (*Referenzfahrtgeschwindigkeit, um Endschalter zu suchen, positive oder negative Werte:1=langsam,2=schnell*)
	REFVEL2:REAL:=-10; (*Referenzfahrtgeschwindigkeit, um vom Endschalter weg die Nullspur zu suchen,  positive oder negative Werte:1=langsam,2=schnel*)
	REF_ON:BOOL; (*Referenzfahrt ohne Nullspur, d.h. bei negtiver Flanke des Endsch. wird Istwert gesetzt*)
	OPTI_KURZ:BOOL;(*optimierung bei kurzer Strecke:Ist der Verfahrweg kleiner als 2*S_SCHLEICH, dann wird auf halbem Weg beschleunugt(EIL) und auf halbem abgebremst (SCHLEICH*)
	WAITTIME_INV:REAL:=0.3;(*Wartezeit bei Richtungsumkehr in SEC*)
	WAIT_Restart_akt:BOOL;(* Wartezeit bei wiederStarten aktiv: wenn der Antrieb abgeschaltet wird, dann bleiben die Ausgänge MINDESTENS "Waittime_INV" abgeschaltet (notwendig bei 24V-DC Lineramotoren) *)
	S_SCHLEICH: REAL;(*Schleichweg*)
	S_STOP: REAL;(*Vorabschaltdifferenz, innerhalb diesem Fenster wird nicht positioniert, sondern PEH ausgegeben!*)
	T_VERZ_STILL:REAL;(*Verzögerungszeit zum Ansprechen der Stillstandsüberwachung, Sekunden*)
	IstWertOffset:LREAL;(*Offset, der  auf den Istwert(Benutzereinheit bzw. mm) Online aufgerechnent wird*)
	MaxIstDiff_pro_Zykl: REAL;(*Einheit: Benutzer (mm) . Wenn zwischen 2 Zyklen eine Istwertänderung (Benutzereinheit bzw. mm) von mehr als dieser Wert auftritt, wird SYNC gelöscht*)
	Loop_val: REAL;		(*schleife fahren: 0=nein; ansonsten: Es wird um den Betrag von S_STOP+Loop_Val vom Ziel weggefahren, abhängig vom Vorzeiche: + in pos.
							Richtung,- in neg. Richtung). Loop_val wird nur bei pos. Flanke Start oder Änderung der Sollpos bei aktivem Start ausgewertet, d.h. eine Änderung während dem Positionieren wird ignoriert*)
END_VAR
VAR_OUTPUT
	DAT_TO_PLC:TES_Achse_IN;(*Übergabe der Parameter zum Anwenderprogramm *)
	COUNT_CTRL: BYTE;(*Verknüpfung mit COUNTER CTRL*)
	EIL_OUT:BOOL;(*Verknüpfung mit Ausgang schnell*)
	VOR_OUT:BOOL;(*Verknüpfung mit Ausgang vor*)
	ZUR_OUT:BOOL;(*Verknüpfung mit Ausgang zur*)
	ERR_INIT:BOOL:=TRUE;(*Fehler bei initialisierung oder noch nicht initialisiert*)
END_VAR

VAR

(*########################################Ausgangsvariabeln vom Baustein -> STRUKTUR(IN) ###################################*)
	IstPos: LREAL;(*Istposition Achse *)
	SYNC: BOOL := FALSE;
	PEH:BOOL;

(*####################################Folgende Daten werden intern berechnet und verwendet#####################################*)
	OFFSET_INC: LREAL;
	COUNT_INC: DINT;(*Zähler-INCREMENTE*)
	COUNT_INC_LAST: DINT;(*Zähler-INCREMENTE des letzten Zyklus, sofern Zähler-Val gültig war*)
	REFSTATUS: INT; (*0=aus,1=suche Endsch;2=Suche neg.Flanke Endsch;3=suche Nullspur,...7=beendet*)
	LAST_COUNT_CTRL: BYTE;
	V_SOLL:REAL;(*Sollgeschwindifkeit, die aufgrund der berechnungen resultiert.V_F_T wird durch V_Soll UND den zulässigen Rampen (zulässige Geschw.-Änderung pro Zyklus) berechnet*)
	Zieldiff_Pos: LREAL;(*POS-Modus: Differenz zum Ziel*)
	Start_Pos_LAST: BOOL;
	SollPos: LREAL;(*Zielposition bei Positionierung*)
	MODULOVAL_INC:REAL;(*Wert in Incrementen für MODULO-Funktion*)
	TIME_VOR: REAL;
	TIME_ZUR: REAL;
	MODULO_ERG: LREAL;
	StartFRG_Pos: BOOL;
	S_SCHLEICH_I: REAL;(*Schleichweg, Intern. Der Wert S_SCHLEICH (VAR_INPUT) wird auf S_SCHLEICH_I kopiert, außer bei optimierung für kurze Strecken *)
	T_STILLST: REAL;(* abgelaufene Stillstandszeit*)
	SetIstPos: BOOL;
	IstPos_LAST: LREAL;
	IstWertOffset_LAST: LREAL;
	Loop_akt: BOOL;(*Schleife-fahren ist aktiv*)
	c_Loop_val: REAL;(* Kopie von LoopVAL*)
END_VAR

SetIstPos:=FALSE;
(*Kontrolle der Parameter*)
IF T_ZYKL<=0 OR IBW<=0 THEN
	ERR_INIT:=TRUE;VOR_OUT:=FALSE;ZUR_OUT:=FALSE;EIL_OUT:=FALSE;RETURN;(*Regelparameter ungültig,Ausgänge abschalten*)
ELSE ERR_INIT:=FALSE;
END_IF
(*###################### ENDE INIT #####################################################*)

DAT_TO_PLC.STILL:=FALSE;(*Stillstand mit FALSE init.*)


(*Zähler auswerten und konvertieren nach INC_IN, wenn RC gesetzt ist: *)
IF C_INVERS THEN COUNT_INC:=16#FFFF-COUNT_VAL;ELSE COUNT_INC:=COUNT_VAL;END_IF
(* Überschläge zählen *)
IF COUNT_INC< 16000 AND COUNT_INC_LAST>48000 THEN OFFSET_INC:=OFFSET_INC+16#10000;(*Überschlag; zum Offset einen COUNTER-Überschlagsbetrag addieren*)
ELSIF COUNT_INC>48000 AND COUNT_INC_LAST<16000 THEN OFFSET_INC:=OFFSET_INC-16#10000;(*Überschlag; vom Offset einen COUNTER-Überschlagsbetrag subtrahieren*)
END_IF



(*Stillstandsüberwachung*)
IF (VOR_OUT AND (COUNT_INC<=COUNT_INC_LAST)) OR (ZUR_OUT AND (COUNT_INC>=COUNT_INC_LAST)) THEN
	T_STILLST:=T_STILLST + T_ZYKL;
	DAT_TO_PLC.STILL:=T_STILLST>T_VERZ_STILL; (*Stillstandsüberwachungszeit abgelaufen ?->SET Stillstand*)
ELSE
	T_STILLST:=0;
END_IF
LAST_COUNT_CTRL:=COUNT_CTRL;

(*############# Referenzmodus: ohne Nullspur oder mit Nullspur ( mit EL,LV COUNTER) #############*)
IF DAT_FROM_PLC.REF THEN
	IF NOT REF_ON THEN (*Referenz mit Nullspur*)
		IF REFSTATUS=0 THEN (*Referenzfahrt hat noch nicht begonnen*)
			SYNC:=FALSE;(*Sync löschen bei Anwahl von Ref-Modus*)
			IF NOT EREF THEN REFSTATUS:=1; (*Refstatus: suche Endschalter*)
			ELSE REFSTATUS:=2; (*Refstatus: Endschalter belegt, suche negative Flanke Endschalter*)
			END_IF
		ELSIF REFSTATUS=1 AND EREF THEN REFSTATUS:=2; (*Wenn Status=suche Endschalter und EREF belegt, dann Status=2*)
		ELSIF REFSTATUS=2 AND NOT EREF THEN REFSTATUS:=3;COUNT_CTRL:=0; (*negative Flanke Endschalter: Nullspur suchen, Status=3, EL  löschen und warten bis L_VALID=0 wird*)
		ELSIF REFSTATUS=3 AND (COUNT_STATE AND 1) = 0 THEN COUNT_CTRL:=1;REFSTATUS:=4;(*LV ist 0, d.h. EL=FALSE wurde angenommen, jetzt muß EL gesetzt werden, damit bei nächster Nullspur LV=1 wird!!!*)
		ELSIF REFSTATUS=4 AND (COUNT_STATE AND 1) <> 0 THEN REFSTATUS:=6; (*LV wurde gültig, jetzt kann  LATCH gelesen werden*)
			(*Offset durch LATCH-Wert neu berechnen*)
			IF C_INVERS THEN OFFSET_INC:=(DAT_FROM_PLC.Refpos/IBW)-(16#FFFF-COUNT_LATCH);COUNT_INC:=DWORD_TO_DINT(16#00FFFF-COUNT_LATCH);
			ELSE OFFSET_INC:=(DAT_FROM_PLC.Refpos/IBW)-COUNT_LATCH;COUNT_INC:=DWORD_TO_DINT(COUNT_LATCH);END_IF
			REFSTATUS:=7;SYNC:=TRUE;SetIstPos:=TRUE;
		END_IF
	ELSE (*Referenz ohne Nullspur*)
		IF REFSTATUS=0 THEN (*Referenzfahrt hat noch nicht begonnen*)
			SYNC:=FALSE;(*Sync löschen bei Anwahl von Ref-Modus*)
			IF NOT EREF THEN REFSTATUS:=1; (*Refstatus: suche Endschalter*)
			ELSE REFSTATUS:=2; (*Refstatus: Endschalter belegt, suche negative Flanke Endschalter*)
			END_IF
		ELSIF REFSTATUS=1 AND EREF THEN REFSTATUS:=2; (*Wenn Status=suche Endschalter und EREF belegt, dann Status=2*)
		ELSIF REFSTATUS=2 AND NOT EREF THEN
			 REFSTATUS:=7; (*negative Flanke Endschalter: Refstatus=7 (fertig, Istwert neu setzen*)
			OFFSET_INC:=DAT_FROM_PLC.RefPos/IBW-COUNT_INC;SYNC:=TRUE;SetIstPos:=TRUE;
		END_IF
	END_IF
ELSE REFSTATUS:=0;COUNT_CTRL:=0; (*Wenn nicht REF-Modus, dann  REFSTATUS=0*)
END_IF
(*MODULOWERT setzen*)
IF DAT_FROM_PLC.MODULO THEN
	IF ABS(COUNT_INC+OFFSET_INC)<16#7FFFFFFF THEN (*MODULO nur möglich, wenn DINT noch nicht erreicht ist*)
		MODULOVAL_INC:=MAX(DAT_FROM_PLC.MODULOVAL_INC,1);(*Div by ZERO!!!*)
		MODULO_ERG:=(LREAL_TO_DINT(COUNT_INC+OFFSET_INC))MOD REAL_TO_DINT (MODULOVAL_INC); (*Modulowert=neuer IstWert*)
		IF MODULO_ERG<0 THEN MODULO_ERG:=MODULO_ERG+MODULOVAL_INC;END_IF
		OFFSET_INC:=MODULO_ERG-COUNT_INC;SetIstPos:=TRUE;(*Offset durch den aktuellen Zählerwert neu berechnen*)
	END_IF

(*Istposition setzen*)
ELSIF DAT_FROM_PLC.SETPOS THEN
	OFFSET_INC:=DAT_FROM_PLC.RefPos/IBW-COUNT_INC;SetIstPos:=TRUE;Sync:=TRUE;
END_IF

(* Ermittlung des Geberistwertes *)
IstPos:=(COUNT_INC+OFFSET_INC)*IBW+IstWertOffset;

IF NOT SetIstPos AND (IstWertOffset=IstWertOffset_LAST) AND ABS(IstPos-IstPos_LAST) > MaxIstDiff_pro_Zykl THEN SYNC:=FALSE;END_IF

(*############################## Achsen-Steuerung ##############################################################*)
PEH:=FALSE; (*PEH mit FALSE initialisieren*)

(*################################ REFERENZFAHRT ################################################*)
IF DAT_FROM_PLC.REF AND NOT SYNC THEN
	IF REFSTATUS=1 THEN V_SOLL:=REFVEL1;
	ELSIF REFSTATUS=7 THEN V_SOLL:=0;
	ELSE V_SOLL:=REFVEL2;
	END_IF

(*########################## Positionieren auf Sollposition######################################*)
(*POSITIONIEREN POSITIONIEREN POSITIONIEREN POSITIONIEREN POSITIONIEREN POSITIONIEREN POSITIONIEREN POSITIONIEREN *)
ELSIF DAT_FROM_PLC.Start_Pos THEN
	Zieldiff_Pos:=DAT_FROM_PLC.Sollpos-IstPos;(*Reelle momentane Differenz zum Ziel*)
	IF NOT Start_Pos_LAST OR Sollpos<>DAT_FROM_PLC.Sollpos THEN (*Flanke Start oder änderung der Sollposition: Werte übergeben*)
		c_Loop_val:=Loop_val; (*Loop-Val speichern, wird während dem Positionieren ignoriert*)
		Loop_akt:=ABS(c_Loop_val) <>0 AND ABS(Zieldiff_Pos)<(S_STOP+ABS(c_Loop_val));
		SollPos:=DAT_FROM_PLC.Sollpos;DAT_TO_PLC.RET_SollPos:=Sollpos;StartFRG_Pos:=TRUE;(*Setzen der Startfreigabe*)
		IF OPTI_KURZ AND ABS(Zieldiff_Pos)<(2*S_SCHLEICH) THEN S_SCHLEICH_I:=LREAL_TO_REAL(ABS(Zieldiff_Pos)/2)+S_STOP;
		ELSE S_SCHLEICH_I:=S_SCHLEICH;
		END_IF
	END_IF

	IF ABS(Zieldiff_Pos)>(S_STOP+ABS(c_Loop_val)) THEN
		Loop_akt:=FALSE;
	END_IF

	IF Loop_akt THEN
		IF StartFRG_Pos THEN
			IF c_Loop_val > 0 THEN (*vorwärts schleife fahren*)
				V_SOLL:=1; (*langsam vor*)
			ELSE (*rückwärts schleife fahren*)
				V_SOLL:=-1; (*langsam zur*)
			END_IF
		ELSE
			V_SOLL:=0; (*keine Startfreigabe (Positionierung bereits ausgeführt), also STOP*)
		END_IF

	ELSIF ABS(Zieldiff_Pos)>S_STOP THEN (*Positionieren, STOP-Fenster noch nicht erreicht*)
		IF StartFRG_Pos THEN
			IF Zieldiff_Pos > 0 THEN (*vorwärts positionieren*)
				IF Zieldiff_Pos > S_SCHLEICH_I AND DAT_FROM_PLC.V_Pos>1 THEN V_SOLL:=2; (*schnell vor*)
				ELSE V_SOLL:=1; (*langsam vor*)
				END_IF
			ELSE (*rückwärts positionieren*)
				IF -Zieldiff_Pos > S_SCHLEICH_I AND DAT_FROM_PLC.V_Pos>1 THEN V_SOLL:=-2; (*schnell zurück*)
				ELSE V_SOLL:=-1; (*langsam zurück*)
				END_IF
			END_IF
		ELSE
			V_SOLL:=0; (*keine Startfreigabe (Positionierung bereits ausgeführt), also STOP*)
		END_IF
	ELSE  (*S_STOP-Fenster bereits erreicht*)
		PEH:=TRUE;
		V_SOLL:=0;
		StartFRG_Pos:=FALSE;
	END_IF


(*################### JOG-Betrieb mit konstanter Geschwindigkeit ohne Startrampe ###################*)
(* JOG JOG JOG JOG JOG JOG JOG JOG JOG JOG JOG JOG JOG JOG JOG JOG JOG JOG JOG JOG JOG JOG JOG JOG JOG JOG JOG *)
ELSIF DAT_FROM_PLC.JOGFW THEN
	V_SOLL:=DAT_FROM_PLC.V_JOG;

ELSIF DAT_FROM_PLC.JOGBW THEN
	V_SOLL:=-DAT_FROM_PLC.V_JOG;

(*####################### Anhalten, keine Bedingung erfüllt##########################################*)
(* HALT HALT HALT HALT HALT HALT HALT HALT HALT HALT HALT HALT HALT HALT HALT HALT HALT HALT HALT HALT HALT HALT *)
ELSE V_SOLL:=0;
END_IF


(*########## Berechnung der Ausgänge ###############*)
IF V_SOLL > 0 THEN (*Sollgeschwindigkeit vor*)
	IF TIME_ZUR=0 AND (TIME_VOR=0 OR  NOT WAIT_Restart_akt OR VOR_OUT) THEN (*keine Richtungsumkehr, rückwärts-Wartezeit ist abgelaufen UND keine wartezeit Restart oder abgelaufen oder fährt bereits*)
		(*positionieren vor*)
		TIME_VOR:=WAITTIME_INV;(*Wartezeit laden*)
		IF V_SOLL=2 THEN DAT_TO_PLC.VEL_IST:=2;
		ELSE DAT_TO_PLC.VEL_IST:=1;
		END_IF
	ELSE (*Rückwärts-Wartezeit läuft noch*)
		DAT_TO_PLC.VEL_IST:=0;
	END_IF
ELSIF V_SOLL < 0 THEN(*Sollgeschwindigkeit negativ*)
	IF TIME_VOR=0 AND (TIME_ZUR=0 OR  NOT WAIT_Restart_akt OR ZUR_OUT) THEN (*keine Richtungsumkehr, vorwärts-Wartezeit ist abgelaufen UND keine wartezeit Restart oder abgelaufen oder fährt bereits*)
		(*positionieren zurück*)
		TIME_ZUR:=WAITTIME_INV;(*Wartezeit "zurück" laden*)
		IF V_SOLL=-2 THEN DAT_TO_PLC.VEL_IST:=-2;
		ELSE DAT_TO_PLC.VEL_IST:=-1;
		END_IF
	ELSE (*vorwärts-Wartezeit läuft noch*)
		DAT_TO_PLC.VEL_IST:=0;
	END_IF
ELSE (*Sollgeschwindigkeit = 0, also STOP*)
	DAT_TO_PLC.VEL_IST:=0;
END_IF
(*Wartezeit decrementieren*)
TIME_VOR:=MAX((TIME_VOR-T_ZYKL),0);TIME_ZUR:=MAX((TIME_ZUR-T_ZYKL),0);
(*Zyklusverz. Var.*)
COUNT_INC_LAST:=COUNT_INC;
Start_Pos_LAST:=DAT_FROM_PLC.Start_Pos;

(*Ausgangsvariablen übergeben*)
DAT_TO_PLC.IstPos:=IstPos;
DAT_TO_PLC.SYNC:=SYNC;
DAT_TO_PLC.PEH:=PEH;
(*Ausgänge setzen*)
VOR_OUT:=DAT_TO_PLC.VEL_IST>0;
ZUR_OUT:=DAT_TO_PLC.VEL_IST<0;
EIL_OUT:=ABS(DAT_TO_PLC.VEL_IST)>=2;
IstPos_Last:=IstPos;
IstWertOffset_LAST:=IstWertOffset;

END_FUNCTION_BLOCK

// POUs/Achsen_Bausteinen/ES_M3120
FUNCTION_BLOCK ES_M3120(*Eil-Schleich - Achse für Encoderbox M3120*)
VAR_INPUT
	DAT_FROM_PLC:TES_Achse_OUT; (*Übergabe der Parameter vom Anwenderprogramm *)
	COUNT_VAL: DINT;(*Verknüpfung mit COUNTER VAL*)
	COUNT_STATE: BYTE;(*Verknüpfung mit COUNTER STATE*)
	EREF: BOOL; (*Verknüpfung mit Referenzeingang*)

(*####################### Folgende Werte sind Regelparameter und müssen initialisiert werden##########################*)
	T_ZYKL: REAL:=0.001;(*Zykluszeit in s, in der dieser Baustein aufgerufen wird*)
	C_INVERS:BOOL:=FALSE; (*Zählrichtungsumkehr*)
	IBW:LREAL:=0.1; (*Istbewertung in mm pro Increment*)
	REFVEL1:REAL:=10; (*Referenzfahrtgeschwindigkeit, um Endschalter zu suchen, positive oder negative Werte:1=langsam,2=schnell*)
	REFVEL2:REAL:=-10; (*Referenzfahrtgeschwindigkeit, um vom Endschalter weg die Nullspur zu suchen,  positive oder negative Werte:1=langsam,2=schnel*)
	REF_ON:BOOL; (*Referenzfahrt ohne Nullspur, d.h. bei negtiver Flanke des Endsch. wird Istwert gesetzt*)
	OPTI_KURZ:BOOL;(*optimierung bei kurzer Strecke:Ist der Verfahrweg kleiner als 2*S_SCHLEICH, dann wird auf halbem Weg beschleunugt(EIL) und auf halbem abgebremst (SCHLEICH*)
	WAITTIME_INV:REAL:=0.3;(*Wartezeit bei Richtungsumkehr in SEC*)
	S_SCHLEICH: REAL;(*Schleichweg*)
	S_STOP: REAL;(*Vorabschaltdifferenz, innerhalb diesem Fenster wird nicht positioniert, sondern PEH ausgegeben!*)
	T_VERZ_STILL:REAL;(*Verzögerungszeit zum Ansprechen der Stillstandsüberwachung, Seckunden*)
	IstWertOffset:LREAL;(*Offset, der  auf den Istwert(Benutzereinheit bzw. mm) Online aufgerechnent wird*)
	MaxIstDiff_pro_Zykl: REAL;(*Einheit: Benutzer (mm). Wenn zwischen 2 Zyklen eine Istwertänderung (Benutzereinheit bzw. mm) von mehr als dieser Wert auftritt, wird SYNC gelöscht*)
END_VAR
VAR_OUTPUT
	DAT_TO_PLC:TES_Achse_IN;(*Übergabe der Parameter zum Anwenderprogramm *)
	COUNT_CTRL: BYTE;(*Verknüpfung mit COUNTER CTRL*)
	EIL_OUT:BOOL;(*Verknüpfung mit Ausgang schnell*)
	VOR_OUT:BOOL;(*Verknüpfung mit Ausgang vor*)
	ZUR_OUT:BOOL;(*Verknüpfung mit Ausgang zur*)
	ERR_INIT:BOOL:=TRUE;(*Fehler bei initialisierung oder noch nicht initialisiert*)
END_VAR

VAR

(*########################################Ausgangsvariabeln vom Baustein -> STRUKTUR(IN) ###################################*)
	IstPos: LREAL;(*Istposition Achse *)
	SYNC: BOOL := FALSE;
	PEH:BOOL;

(*####################################Folgende Daten werden intern berechnet und verwendet#####################################*)
	OFFSET_INC: LREAL;
	COUNT_INC: DINT;(*Zähler-INCREMENTE*)
	COUNT_INC_LAST: DINT;(*Zähler-INCREMENTE des letzten Zyklus, sofern Zähler-Val gültig war*)
	REFSTATUS: INT; (*0=aus,1=suche Endsch;2=Suche neg.Flanke Endsch;3=suche Nullspur,...7=beendet*)
	LAST_COUNT_CTRL: BYTE;
	V_SOLL:REAL;(*Sollgeschwindifkeit, die aufgrund der berechnungen resultiert.V_F_T wird durch V_Soll UND den zulässigen Rampen (zulässige Geschw.-Änderung pro Zyklus)berechnet*)
	Zieldiff_Pos: LREAL;(*POS-Modus: Differenz zum Ziel*)
	Start_Pos_LAST: BOOL;
	SollPos: LREAL;(*Zielposition bei Positionierung*)
	MODULOVAL_INC:REAL;(*Wert in Incrementen für MODULO-Funktion*)
	TIME_VOR: REAL;
	TIME_ZUR: REAL;
	MODULO_ERG: LREAL;
	StartFRG_Pos: BOOL;
	S_SCHLEICH_I: REAL;(*Schleichweg, Intern. Der Wert S_SCHLEICH (VAR_INPUT) wird auf S_SCHLEICH_I kopiert, außer bei optimierung für kurze Strecken *)
	T_STILLST: REAL;(* abgelaufene Stillstandszeit*)
	SetIstPos: BOOL;
	IstPos_LAST: LREAL;
END_VAR

SetIstPos:=FALSE;
(*Kontrolle der Parameter*)
IF T_ZYKL<=0 OR IBW<=0 THEN
	ERR_INIT:=TRUE;VOR_OUT:=FALSE;ZUR_OUT:=FALSE;EIL_OUT:=FALSE;RETURN;(*Regelparameter ungültig,Ausgänge abschalten*)
ELSE ERR_INIT:=FALSE;
END_IF
(*###################### ENDE INIT #####################################################*)

DAT_TO_PLC.STILL:=FALSE;(*Stillstand mit FALSE init.*)


(*Zähler auswerten und konvertieren nach INC_IN, wenn RC gesetzt ist: *)
IF (COUNT_CTRL AND 1) <> 0 AND (LAST_COUNT_CTRL AND 1) <> 0 THEN(* Zähler ist gültig, Istwerte werden ausgelesen*)
	(* Zähler invertieren wenn INV=1*)
	IF C_INVERS THEN COUNT_INC:=16#00FFFFFF-COUNT_VAL;ELSE COUNT_INC:=COUNT_VAL;END_IF
	(* Überschläge zählen *)
	IF COUNT_INC<4000000 AND COUNT_INC_LAST>12000000 THEN OFFSET_INC:=OFFSET_INC+16#1000000;(*Überschlag; zum Offset einen COUNTER-Überschlagsbetrag addieren*)
	ELSIF COUNT_INC>12000000 AND COUNT_INC_LAST<4000000 THEN OFFSET_INC:=OFFSET_INC-16#1000000;(*Überschlag; vom Offset einen COUNTER-Überschlagsbetrag subtrahieren*)
	END_IF
	(*Stillstandsüberwachung*)
	IF (VOR_OUT AND (COUNT_INC<=COUNT_INC_LAST)) OR (ZUR_OUT AND (COUNT_INC>=COUNT_INC_LAST)) THEN
		T_STILLST:=T_STILLST + T_ZYKL;
		DAT_TO_PLC.STILL:=T_STILLST>T_VERZ_STILL; (*Stillstandsüberwachungszeit abgelaufen ?->SET Stillstand*)
	ELSE
		T_STILLST:=0;
	END_IF
END_IF
LAST_COUNT_CTRL:=COUNT_CTRL;



(*############# Referenzmodus: ohne Nullspur oder mit Nullspur ( mit EL,LV COUNTER) #############*)
IF DAT_FROM_PLC.REF THEN
	IF NOT REF_ON THEN (*Referenz mit Nullspur*)
		IF REFSTATUS=0 THEN (*Referenzfahrt hat noch nicht begonnen*)
			SYNC:=FALSE;(*Sync löschen bei Anwahl von Ref-Modus*)
			IF NOT EREF THEN REFSTATUS:=1; (*Refstatus: suche Endschalter*)
			ELSE REFSTATUS:=2; (*Refstatus: Endschalter belegt, suche negative Flanke Endschalter*)
			END_IF
		ELSIF REFSTATUS=1 AND EREF THEN REFSTATUS:=2; (*Wenn Status=suche Endschalter und EREF belegt, dann Status=2*)
		ELSIF REFSTATUS=2 AND NOT EREF THEN REFSTATUS:=3;COUNT_CTRL:=9; (*negative Flanke Endschalter: Nullspur suchen, Status=3, RC und EL setzten*)
		ELSIF REFSTATUS=3 AND (COUNT_STATE AND 32) = 0 THEN COUNT_CTRL:=1;REFSTATUS:=4;(*LV ist 0, d.h. EL wurde angenommen, jetzt muß EL gelöscht werden, damit bei nächster Nullspur LV=1 wird!!!*)
		ELSIF REFSTATUS=4 AND (COUNT_STATE AND 32) <> 0 THEN COUNT_CTRL:=2;REFSTATUS:=5; (*LV wurde gültig, jetzt READ LATCH setzen: RL=1,RC=0*)
		ELSIF REFSTATUS=5 THEN REFSTATUS:=6; (* Einen Zyklus warten, LATCH-Wert wird erst im nächsten Zyklus gültig*)
		ELSIF REFSTATUS=6 THEN (*Offset durch LATCH-Wert neu berechnen*)
			IF C_INVERS THEN OFFSET_INC:=(DAT_FROM_PLC.Refpos/IBW)-(16#00FFFFFF-COUNT_VAL);ELSE OFFSET_INC:=(DAT_FROM_PLC.Refpos/IBW)-COUNT_VAL;END_IF
			COUNT_CTRL:=1;REFSTATUS:=7;SYNC:=TRUE;SetIstPos:=TRUE;
		END_IF
	ELSE (*Referenz ohne Nullspur*)
		IF REFSTATUS=0 THEN (*Referenzfahrt hat noch nicht begonnen*)
			SYNC:=FALSE;(*Sync löschen bei Anwahl von Ref-Modus*)
			IF NOT EREF THEN REFSTATUS:=1; (*Refstatus: suche Endschalter*)
			ELSE REFSTATUS:=2; (*Refstatus: Endschalter belegt, suche negative Flanke Endschalter*)
			END_IF
		ELSIF REFSTATUS=1 AND EREF THEN REFSTATUS:=2; (*Wenn Status=suche Endschalter und EREF belegt, dann Status=2*)
		ELSIF REFSTATUS=2 AND NOT EREF THEN
			 REFSTATUS:=7; (*negative Flanke Endschalter: Refstatus=7 (fertig, Istwert neu setzen*)
			OFFSET_INC:=DAT_FROM_PLC.RefPos/IBW-COUNT_INC;SYNC:=TRUE;SetIstPos:=TRUE;
		END_IF
	END_IF
ELSE REFSTATUS:=0;COUNT_CTRL:=1; (*Wenn nicht REF-Modus, dann RC setzen, REFSTATUS=0*)
END_IF

(*MODULOWERT setzen*)
IF DAT_FROM_PLC.MODULO THEN
	IF ABS(COUNT_INC+OFFSET_INC)<16#7FFFFFFF THEN (*MODULO nur möglich, wenn DINT noch nicht erreicht ist*)
		MODULOVAL_INC:=MAX(DAT_FROM_PLC.MODULOVAL_INC,1);(*Div by ZERO!!!*)
		MODULO_ERG:=(LREAL_TO_DINT(COUNT_INC+OFFSET_INC))MOD REAL_TO_DINT (MODULOVAL_INC); (*Modulowert=neuer IstWert*)
		IF MODULO_ERG<0 THEN MODULO_ERG:=MODULO_ERG+MODULOVAL_INC;END_IF
		OFFSET_INC:=MODULO_ERG-COUNT_INC;SetIstPos:=TRUE;(*Offset durch den aktuellen Zählerwert neu berechnen*)
	END_IF

(*Istposition setzen*)
ELSIF DAT_FROM_PLC.SETPOS THEN
	OFFSET_INC:=DAT_FROM_PLC.RefPos/IBW-COUNT_INC;SetIstPos:=TRUE;Sync:=TRUE;
END_IF

(* Ermittlung des Geberistwertes *)
IstPos:=(COUNT_INC+OFFSET_INC)*IBW+IstWertOffset;

IF NOT SetIstPos AND ABS(IstPos-IstPos_LAST) > MaxIstDiff_pro_Zykl THEN SYNC:=FALSE;END_IF


(*############################## Achsen-Steuerung ##############################################################*)
PEH:=FALSE; (*PEH mit FALSE initialisieren*)

(*################################ REFERENZFAHRT ################################################*)
IF DAT_FROM_PLC.REF AND NOT SYNC THEN
	IF REFSTATUS=1 THEN V_SOLL:=REFVEL1;
	ELSIF REFSTATUS=7 THEN V_SOLL:=0;
	ELSE V_SOLL:=REFVEL2;
	END_IF

(*########################## Positionieren auf Sollposition######################################*)
(*POSITIONIEREN POSITIONIEREN POSITIONIEREN POSITIONIEREN POSITIONIEREN POSITIONIEREN POSITIONIEREN POSITIONIEREN *)
ELSIF DAT_FROM_PLC.Start_Pos THEN
	Zieldiff_Pos:=DAT_FROM_PLC.Sollpos-IstPos;(*Reelle momentane Differenz zum Ziel*)
	IF NOT Start_Pos_LAST OR Sollpos<>DAT_FROM_PLC.Sollpos THEN (*Flanke Start oder änderung der Sollposition: Werte übergeben*)
		SollPos:=DAT_FROM_PLC.Sollpos;DAT_TO_PLC.RET_SollPos:=Sollpos;StartFRG_Pos:=TRUE;(*Setzen der Startfreigabe*)
		IF OPTI_KURZ AND ABS(Zieldiff_Pos)<(2*S_SCHLEICH) THEN S_SCHLEICH_I:=LREAL_TO_REAL(ABS(Zieldiff_Pos)/2)+S_STOP;
		ELSE S_SCHLEICH_I:=S_SCHLEICH;
		END_IF
	END_IF
	IF ABS(Zieldiff_Pos)>S_STOP THEN (*Positionieren, STOP-Fenster noch nicht erreicht*)
		IF StartFRG_Pos THEN
			IF Zieldiff_Pos > 0 THEN (*vorwärts positionieren*)
				IF Zieldiff_Pos > S_SCHLEICH_I AND DAT_FROM_PLC.V_Pos>1 THEN V_SOLL:=2; (*schnell vor*)
				ELSE V_SOLL:=1; (*langsam vor*)
				END_IF
			ELSE (*rückwärts positionieren*)
				IF -Zieldiff_Pos > S_SCHLEICH_I AND DAT_FROM_PLC.V_Pos>1 THEN V_SOLL:=-2; (*schnell zurück*)
				ELSE V_SOLL:=-1; (*langsam zurück*)
				END_IF
			END_IF
		ELSE
			V_SOLL:=0; (*keine Startfreigabe (Positionierung bereits ausgeführt), also STOP*)
		END_IF
	ELSE  (*S_STOP-Fenster bereits erreicht*)
		PEH:=TRUE;
		V_SOLL:=0;
		StartFRG_Pos:=FALSE;
	END_IF


(*################### JOG-Betrieb mit konstanter Geschwindigkeit ohne Startrampe ###################*)
(* JOG JOG JOG JOG JOG JOG JOG JOG JOG JOG JOG JOG JOG JOG JOG JOG JOG JOG JOG JOG JOG JOG JOG JOG JOG JOG JOG *)
ELSIF DAT_FROM_PLC.JOGFW THEN
	V_SOLL:=DAT_FROM_PLC.V_JOG;

ELSIF DAT_FROM_PLC.JOGBW THEN
	V_SOLL:=-DAT_FROM_PLC.V_JOG;

(*####################### Anhalten, keine Bedingung erfüllt##########################################*)
(* HALT HALT HALT HALT HALT HALT HALT HALT HALT HALT HALT HALT HALT HALT HALT HALT HALT HALT HALT HALT HALT HALT *)
ELSE V_SOLL:=0;
END_IF


(*########## Berechnung der Ausgänge ###############*)
IF V_SOLL > 0 THEN (*Sollgeschwindigkeit vor*)
	IF TIME_ZUR=0 THEN (*keine Richtungsumkehr, rückwärts-Wartezeit ist abgelaufen*)
		(*positionieren vor*)
		TIME_VOR:=WAITTIME_INV;(*Wartezeit laden*)
		IF V_SOLL=2 THEN DAT_TO_PLC.VEL_IST:=2;
		ELSE DAT_TO_PLC.VEL_IST:=1;
		END_IF
	ELSE (*Rückwärts-Wartezeit läuft noch*)
		DAT_TO_PLC.VEL_IST:=0;
	END_IF
ELSIF V_SOLL < 0 THEN(*Sollgeschwindigkeit negativ*)
	IF TIME_VOR=0 THEN (*keine Richtungsumkehr, vorwärts-Wartezeit ist abgelaufen*)
		(*positionieren zurück*)
		TIME_ZUR:=WAITTIME_INV;(*Wartezeit "zurück" laden*)
		IF V_SOLL=-2 THEN DAT_TO_PLC.VEL_IST:=-2;
		ELSE DAT_TO_PLC.VEL_IST:=-1;
		END_IF
	ELSE (*vorwärts-Wartezeit läuft noch*)
		DAT_TO_PLC.VEL_IST:=0;
	END_IF
ELSE (*Sollgeschwindigkeit = 0, also STOP*)
	DAT_TO_PLC.VEL_IST:=0;
END_IF
(*Wartezeit decrementieren*)
TIME_VOR:=MAX((TIME_VOR-T_ZYKL),0);TIME_ZUR:=MAX((TIME_ZUR-T_ZYKL),0);
(*Zyklusverz. Var.*)
COUNT_INC_LAST:=COUNT_INC;
Start_Pos_LAST:=DAT_FROM_PLC.Start_Pos;

(*Ausgangsvariablen übergeben*)
DAT_TO_PLC.IstPos:=IstPos;
DAT_TO_PLC.SYNC:=SYNC;
DAT_TO_PLC.PEH:=PEH;
(*Ausgänge setzen*)
VOR_OUT:=DAT_TO_PLC.VEL_IST>0;
ZUR_OUT:=DAT_TO_PLC.VEL_IST<0;
EIL_OUT:=ABS(DAT_TO_PLC.VEL_IST)>=2;
IstPos_Last:=IstPos;

END_FUNCTION_BLOCK

// POUs/Achsen_Bausteinen/KR_Achse_V2
FUNCTION_BLOCK KR_Achse_V2 (*Kontinuierliche, Ruckbegrenzte Achse V2
Version: 2.01	29.09.2014	Walter Lanz 
	V2.02	(6.10.2014)
		Adapter füR Encodersimulation angepas, Parameterbeschreibungen

	V2.03 (7.10.2014, LanWal)
		Achse um INPUT SIMULATION erweitert (Encodersimulation)
		Adapter füR Encodersimulation gelöscht
		Berechnungen füR Achs_IN.BrakingDist, Achs_IN.BrakingTime und Achs_IN.PosTime füR
		nicht Ruckbegrenztes positionieren implementiert.

	V2.04 (19.6.2015, LanWal)
		-Kommentar bei IBW2 richtiggestellt: 10 0000H Incremente/Motorumdrehung bei EnDat
		-FUNCTION_BLOCK Adapter_Drive_MDS geändert: für IPM-Modus erweitert, für externen Encoder ( IPM-Modus wenn der Geber zur Istwerterfassung NICHT der Motorgeber ist,  z.B. Achse Vorschub oder Positionsmessung mit Laser ) oder ohne Ex. Encoder prametrierbar 
		geänderte Module:
			-KR_Achse_V2.Regelung
			-KR_Achse_V2
			-FUNCTION_BLOCK Adapter_Drive_MDS
			-TYPE TAchs_To_DriveAdapter

	V2.05 (6.7.2015, LanWal): Bei Istwertsprung der grösser als "Istwertsprung_f_RstSync" ist, wird SYNC gelöscht. Nur für Incrementalachsen relevant.

	V2.06: (20.2.16 LanWal):
		B1ugfix1: Bremsrampe wird nicht übernommen in Bremsphase bei Wechsel von Ruckbegr.Positionierung zu Positionierung ohne Ruckbegrenzung. 
						Das Ziel wird dabei eventuell überfahren)
		Bugfix2: Referenz wird bei incrementalachsen nie ausgeführt da sich diese selber löscht wegen istwertsprung; fehlende Konvertierung DWord_to_dint.			

	V2.07: (22.2.16 LanWal):
		Schleppabstand löschen bei Counter-Überschlag (Istwertüberschlag) bei Absolutachsen. (z.b. bei Verwendung als Moduloachse sinnvoll). Funktioniert aber nicht.

	V2.08: (23.2.16 LanWal):
		BugFIX beim: Schleppabstand löschen bei Counter-Überschlag (Istwertüberschlag) bei Absolutachsen. (z.b. bei Verwendung als Moduloachse sinnvoll)

	V2.09: (24.3.16 LanWal):
		BugFix : Sync wird gelöscht wenn Incrementalachse und counter_bits<32.

	V2.10: (6.4.16 ) Adapter von Pitscheider Oswald "lengendärer Ossi" eingefügt: FUNCTION_BLOCK Adapter_Drive_BeckhoffEL7201 Adapter für Beckhoff Servomotorklemme EL7201

	V2.11: (30.05.17 priphi) Adapter für SI6 Umrichter "Adapter_Drive_SI6" und PDO IO Strukturen eingefügt.

	V2.12: Adapter für Analogklemme eingefügt von UNBEKANNT

	V2.13: (04.08.17 lanwal): Bugfix Aufgrund vom Chrash bei Regenold SPR durch Überspannung aufgedeckt. BUG:
		Wenn im Positioniermodus in Fase 4,5 oder 6 Start_Pos weggenommen wird, übernimmt die Achse fälschlicherweise die Bremsbeschleunigung "DCC_JRS" wenn sie 
		kleiner als die  ursprüngliche DCC_Pos ist. Die Folge ist ein nicht Ruckbegrenztes abbremsen durch Err_ID=12, da die übernommene Bremsrampe ein Überfahren des Zieles zur 
		Folge hätte. Änderung in FUNCTION_BLOCK Phase56 / 8 (Abfrage GT anstatt LE).
	
	V2.14: (9.10.17 lanwal): Die Variablen Achs_IN.BrakingDist, BrakingTime und Postime wurden beim Positionieren OHNE Ruckbegrenzung (RB=0) falsch berechnet, es wurde 
		die Achs_OUT.DCC_JRS zur Berechnung herangezogen anstatt DCC_POS. (KR_Achse_VS /53+54 )

	V2.15: 109.10.17 lanwal):
		 Bugfix1: bei Wegnahme von Start wird in Achs_IN.Postime jetzt der Wert -1 (unbekannt) zurückgemeldet (Vorher wurde die Bremszeit übergeben was zu Fehlverhalten im Anwenderporgramm führen kann.
		 Bugfix2: Achs_IN.Postime wurde bis V2.14 nur beim vorwärtsfahren ab Phase 4 berechnet, beim rückwärtsfahren erst ab Phase 5. Jetzt wird für beide Richtungen bis Phase 4 der Wert -1 (unbekannt) zurückgemeldet, 
			ab Phase 4 die effektive Positionierzeit

	V2.17: nicht verwenden! 

	V2.18: 21.02.18 (lanwal): Aufgrund des Fehlers Err_ID=13, da Phase 7 nicht eingeleitet und eine Richtungsumkehr erkannt wurde, Fehler ist bei Srob Jungwirth aufgefallen, der Fehler trat bei einem Positionierweg von 0,000055 mm auf:
	Das Problem war, dass IV_RB.HalfCyklVelDiff=0 war, da sich die Achse zuletzt in Phase 4 befand, durch einleiten der Phase 5 kam es aber zur Richtungsumkehr.
	Änderung: Phase56 / 11 

	V2.19. ?

	V2.20: 30.8.2018 (WLA) "Adapter_DriveBased_U" eingefügt: universaladapter für Drivebased-Antriebe

	V2.21: 18.2.2019 (walpet) "Phase7 NW10 Sel geändert Nur für TwinCat 3 relevant

	V2.23: 18.2.2019 (walpet) Adapter V3 und Limitierung IstOffset eingefügt
	
	V2.23.0.3: 31.1.2020 (niest2) Encodersimulation Limitierung auf DINT Wertebereich korrigiert
	
	V2.23.0.4:	03.09.2020 (niest2) Adapter Beckhoff EL7201 Konvertierung richtig gestellt

	V2.23.0.5:	08.03.2021 (niest2): FB ES_EL5xx1_A hinzugefügt: Eil-Schleich Achse für Encoderklemmen, verfügbare Counter Bits können übergeben werden 	

	V2.23.0.7:	2024-04 (WLA) Bugfix falsch berechneter Brensweg bei Wegnahme von Start in Phase 6.
	
*)

VAR_INPUT
	Achs_CMD:TKont_Achse_OUT; (*Übergabe der Parameter vom Anwenderprogramm *)
	CounterVal: DINT;		(*Verknüpfung mit COUNTER VAL. Folgende Typen können Parametriert werden: WORD,INT,DWORD,DINT*)
	counter_bits:INT:=32;(*Anzahl der Bits die ein Counter verwendet.
	Incrementalgeber: Es können weniger als die zu Verfügung stehenden Bits des Encoders angegeben werden, es dürfen aber niemals mehr als die zu Verfügung stehenden Bits des Encoders angegeben werden
			da ansonsten der Überschlag nicht erkannt wird und somit sehr hohe Istwertsprünge auftreten und der Istwert ungültig wird
	Absolutgeber:  Es können weniger als die zu Verfügung stehenden Bits des Encoders angegeben werden (dabei wird aber nicht der volle mögliche Zählweg genutzt ), es dürfen aber niemals mehr als
			die zu Verfügung stehenden Bits des Encoders angegeben werden.  Es sollte immer Kontrolliert werden, daß der Gesamtweg NICHT die Multiturn-Anzahl der Drehgebers überschreitet! Die maximale Anzahl der möglichen
			Umdrehungen bei Stöber MDS n-Dat ist 4096 Umdrehungen. Der maximal mögliche  Verfahrweg ist (mm/Umdr)*4096 *)
	EREF: BOOL;(*Verknüpfung mit Referenzeingang*)
(*####################### Folgende Werte sind Regelparameter und müssen initialisiert werden##########################*)
	T_ZYKL: REAL:=0.001;(*Zykluszeit in s, in der dieser Baustein aufgerufen wird*)
	mm_pro_MotUmdr:LREAL:=100; (* für die Berechnung der Bezugsgeschwindigkeit:  mm/ Motorundrehung.
		Umrechnung  von  KR_MDS_ETHERCAT : mm_pro_MotUmdr=V_BEZ/50 (wenn Umrichter auf 3000Upm parametriert war) *)
	KV2: LREAL:=0.2;(*KV-Faktor. Der Faktor bestimmt die Geschwindigkeit / digit, mit der die Lageregelung reagiert. Beispiel: KV=5, Schleppabstand=10mm -> V_regel=5*10=50mm/s
		Umrechnung  von  KR_MDS_ETHERCAT :KV2=KV/100*V_BEZ.*)
	PEH_Fenster:LREAL:=5;(*PEH-Fenster: Bei Positionierung und Referenzfahrt nach erreichen des Referenzpunktes. PEH wird erst im Stillstand (VEL_IST=0) ausgegeben!*)
	Antrieb_INVERS:BOOL; (*Zählrichtung und Sollwert arbeieten invers. soll nur der counterval invertiert werden, kann dem CounterVal ein "-" vorangestellt werden.
	Soll nur der Sollwert invertiert werden, kann die maximaldrehzahl am Adapter (Adapter_Drive_XXXX) negativ angegeben werden, alternativ kann dem CounterVal ein "-" vorangestellt und Antrieb_INVERS=true gesetzt werden*)
	IBW2:LREAL:=0.1; (*Istbewertung in mm pro Increment. Die Angabe ist für Incrementalgeber und Absolutgeber identisch, d.h. es wird NICHT, wie bei KR_MDS_ETHERCAT, für Absolutgeber (EnDat) ein Viertel  der vom Umrichter gelieferten Auflösung angegeben!
					 EnDat: 10 0000 H Incremente / Motorumdrehung
					 Incrementalgeber: Die Counter werten im Normalfall immer die Flanken der Rechtecksignale aus, d.h. die Incrementezahl/Geberumdrehung ist das 4-Fach der Auflösung welche am Typenschild des Drehgebers angegeben ist*)
	REFVEL1: LREAL:=10; (*Referenzfahrtgeschwindigkeit, um Endschalter zu suchen, positive oder negative Werte*)
	REFVEL2: LREAL:=-10; (*Referenzfahrtgeschwindigkeit, um vom Endschalter weg die Nullspur zu suchen,  positive oder negative Werte*)
	KV2_LIMIT: LREAL := 20.0;	(*Limit für den Lageregler.  Einheit in Geschwindigkeit/Wegfehler (mm/s).  Umrechnung  von  KR_MDS_ETHERCAT :KV2_Limit=KV_Limit/100*V_BEZ.*)
	KD2: REAL;		(*Konstante Differenzialverstärkungsfaktor in (mm/s)/(mm/s^2). Umrechnung  von  KR_MDS_ETHERCAT:  KD2=KD/10*V_BEZ *)
	SET_P_T: BOOL; (*setze dierekt P_T, die Achse folgt der vorgegebenen "P_T_VALUE" und "V_T_VALUE"*)
	P_T_VALUE: LREAL;
	V_T_VALUE: LREAL;
	Incrementalgeber: BOOL;	(*	Achse hat Incrementalgeber / false=Absolutgeber *)
	IWTyp:LREAL;(*Istwert Typisch, nur Absolutachse: Dieser Wert ist Notwendig, um den Geberüberschlag intern ausserhalb dem typischen Istwert zu verschieben, er kann
				 mit0 (oder gar nicht = 0) parametriert werden. Nur in Sonderfällen, wo aufgrund einem hohen Verfahrweg der gesamte Geberbereich abgefahren wird, kann es notwendig sein, einen korrekten Wert anzugeben. In 
				diesem fall ist der Mittelwert zwischen Minpos und Maxpos anzugeben; eine Achse, die in diesem Fall z.B. von +20000mm bis +60000 mm verfährt, muss dann mit +40000 parametriert werden. Die maximale Anzahl der möglichen
				Umdrehungen bei Stöber MDS n-Dat ist 4096 Umdrehungen. Der maximal mögliche  Verfahrweg ist (mm/Umdr)*4096 *)
	Simulation: BOOL;
	Istwertsprung_f_RstSync:REAL:=100;(*Ergibt sich zwischen 2 Zyklen ein Istwertsprung (Benutzereinheit: mm...) der höher als Istwertsprung_f_RstSync ist, wird Achs_IN.Sync zurückgesetzt (nur relevant für Incrementalachsen*)
END_VAR
VAR_OUTPUT
	Achs_to_DriveAdapter:TAchs_To_DriveAdapter;
	Achs_State:TKont_Achse_IN; (*Übergabe der Parameter zum Anwenderprogramm *)
END_VAR

VAR
	copy_Counter: DWORD;		(*Zähler-INCREMENTE*)
	REFSTATUS: INT; (*0=aus,1=suche Endsch;2=Suche neg.Flanke Endsch;3=suche Nullspur,...7=beendet*)
	Set_PT_Eq_Istpos: BOOL;(*Achsenzustand einfrieren, z.B. bei ungültigem Istwert (bei Referenzfahrt, bei MODULOWERT...):Analogsignal bleibt unverändert,Schleppabastand wird gelöscht*)
	(*Interne Variablen für Positionieren mit Ruckbegrenzung*)
	KV_ANTEIL: LREAL;
	IstWertOffset_LAST: LREAL;
	D_Anteil: REAL;
	IWT_Offset: DINT;(*Offset für Istwert-Typisch (Absolutachse)*)

	Phase0: Phase0;
	Phase3: Phase3;
	Phase4: Phase4;
	IV_RB: TIV_RB;
	switchPhase: switchPhase;
	Phase12: Phase12;
	Phase56: Phase56;
	Phase7: Phase7;
	MEM_MaxAccubrn: LREAL;
	MEM_MaxDccubrn: LREAL;
	NotBremsWeg: LREAL;
	Abbrch_RB: BOOL;		(*abbruch der Ruckbegrenzung wegen P_T manipulation, reffahrt, Reset ...*)
	V_SOLL: LREAL;
	Sollpos: LREAL;
	V_POS: LREAL;
	ACC_POS: LREAL;
	DCC_POS_oRB: LREAL;
	DCC_STOP_oRB: LREAL;
	CD1_ErrId: CDLR;
	PEH_Val: LREAL;
	PEV_Val: LREAL;
	Zieldiff_Pos: LREAL;
	MEM_MaxGrenzpos: LREAL;
	MEM_MinGrenzpos: LREAL;
	WayError_Fkt: LREAL;
	WayError: LREAL;
	Acc_ist: LREAL;
	BWCycl1: Bremsweg;
	BWCycl2: Bremsweg;
	copy_Counter_Last: DWORD;
	Incr_Offset: LREAL;(*Offset ebi Incremental-counter*)
	EncBitMask: DWORD;
	CountLimit1: DWORD;
	CountLimit2: DWORD;
	Bremsweg_Jog: LREAL;
	Sim_EncoderVal: LREAL;
	TempDint1: DINT;
	TempDint2: DINT;
	EmptyBits: INT;
END_VAR
VAR // added by the converter: edge detectors and wires of the graphical bodies
    _w1 : BOOL;
    _w2, _w3, _w4, _w5, _w7 : LREAL;
    _w6, _w8 : INT;
END_VAR

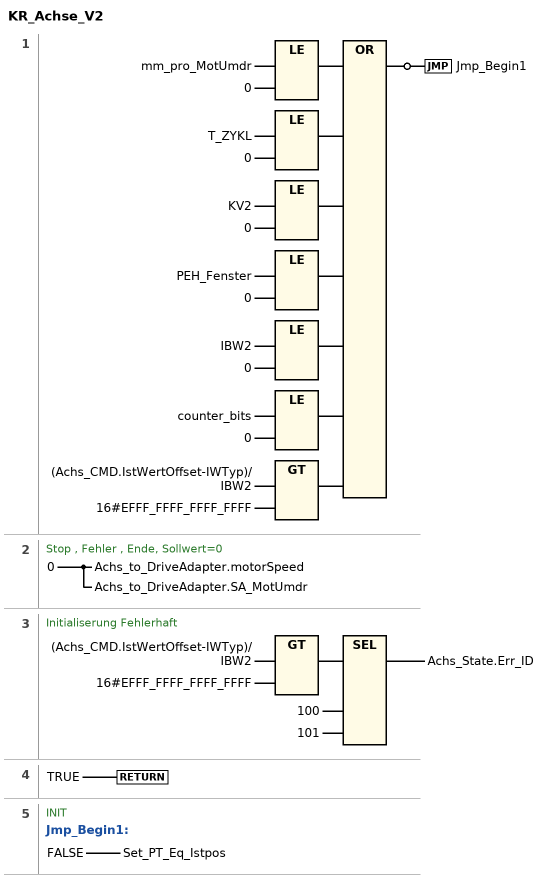
// NETWORK 1
IF NOT (mm_pro_MotUmdr <= 0 OR T_ZYKL <= 0 OR KV2 <= 0 OR PEH_Fenster <= 0 OR IBW2 <= 0 OR counter_bits <= 0 OR ((Achs_CMD.IstWertOffset-IWTyp)/IBW2) > 16#EFFF_FFFF_FFFF_FFFF) THEN JMP Jmp_Begin1; END_IF

// NETWORK 2
// Stop , Fehler , Ende, Sollwert=0
Achs_to_DriveAdapter.motorSpeed := 0;
Achs_to_DriveAdapter.SA_MotUmdr := 0;

// NETWORK 3
// Initialiserung Fehlerhaft
Achs_State.Err_ID := SEL(((Achs_CMD.IstWertOffset-IWTyp)/IBW2) > 16#EFFF_FFFF_FFFF_FFFF, 100, 101);

// NETWORK 4
RETURN;

// NETWORK 5
// INIT
Jmp_Begin1:
Set_PT_Eq_Istpos := FALSE;

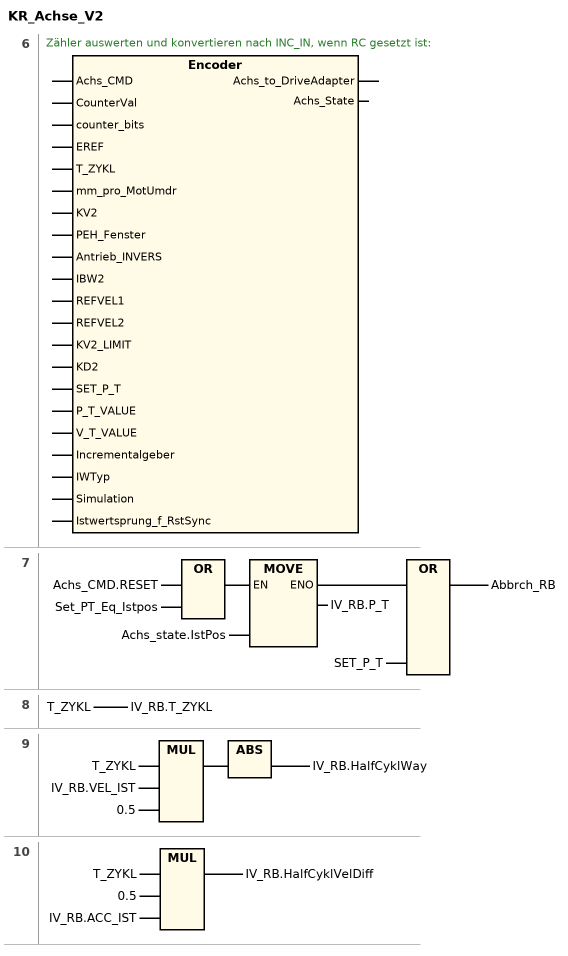
// NETWORK 6
// Zähler auswerten und konvertieren nach INC_IN, wenn RC gesetzt ist:
Encoder();

// NETWORK 7
_w1 := Achs_CMD.RESET OR Set_PT_Eq_Istpos;
IF _w1 THEN IV_RB.P_T := Achs_state.IstPos; END_IF
Abbrch_RB := _w1 OR SET_P_T;

// NETWORK 8
IV_RB.T_ZYKL := T_ZYKL;

// NETWORK 9
IV_RB.HalfCyklWay := ABS(T_ZYKL * IV_RB.VEL_IST * 0.5);

// NETWORK 10
IV_RB.HalfCyklVelDiff := T_ZYKL * 0.5 * IV_RB.ACC_IST;

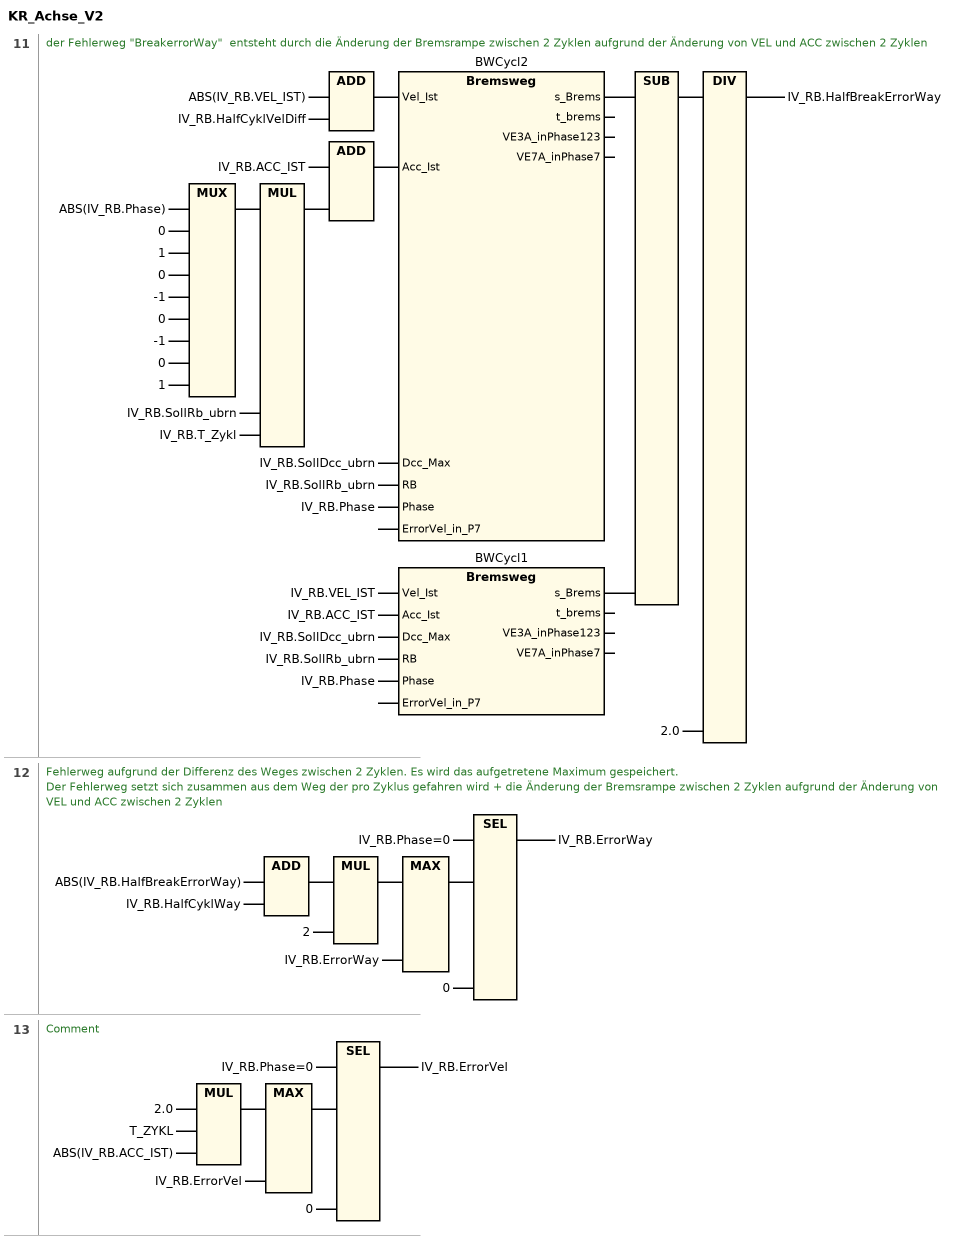
// NETWORK 11
// der Fehlerweg "BreakerrorWay"  entsteht durch die Änderung der Bremsrampe zwischen 2 Zyklen aufgrund der Änderung von VEL und ACC zwischen 2 Zyklen
BWCycl2(
    Vel_Ist := (ABS(IV_RB.VEL_IST)) + IV_RB.HalfCyklVelDiff,
    Acc_Ist := IV_RB.ACC_IST + MUX(ABS(IV_RB.Phase), 0, 1, 0, -1, 0, -1, 0, 1) * IV_RB.SollRb_ubrn * IV_RB.T_Zykl,
    Dcc_Max := IV_RB.SollDcc_ubrn,
    RB := IV_RB.SollRb_ubrn,
    Phase := IV_RB.Phase); // Bremsweg
BWCycl1(
    Vel_Ist := IV_RB.VEL_IST,
    Acc_Ist := IV_RB.ACC_IST,
    Dcc_Max := IV_RB.SollDcc_ubrn,
    RB := IV_RB.SollRb_ubrn,
    Phase := IV_RB.Phase); // Bremsweg
IV_RB.HalfBreakErrorWay := (BWCycl2.s_Brems - BWCycl1.s_Brems) / 2.0;

// NETWORK 12
// 					Fehlerweg aufgrund der Differenz des Weges zwischen 2 Zyklen. Es wird das aufgetretene Maximum gespeichert.
// Der Fehlerweg setzt sich zusammen aus dem Weg der pro Zyklus gefahren wird + die Änderung der Bremsrampe zwischen 2 Zyklen aufgrund der Änderung von VEL und ACC zwischen 2 Zyklen
//
IV_RB.ErrorWay := SEL(IV_RB.Phase=0, MAX(((ABS(IV_RB.HalfBreakErrorWay)) + IV_RB.HalfCyklWay) * 2, IV_RB.ErrorWay), 0);

// NETWORK 13
// Comment
IV_RB.ErrorVel := SEL(IV_RB.Phase=0, MAX(2.0 * T_ZYKL * (ABS(IV_RB.ACC_IST)), IV_RB.ErrorVel), 0);

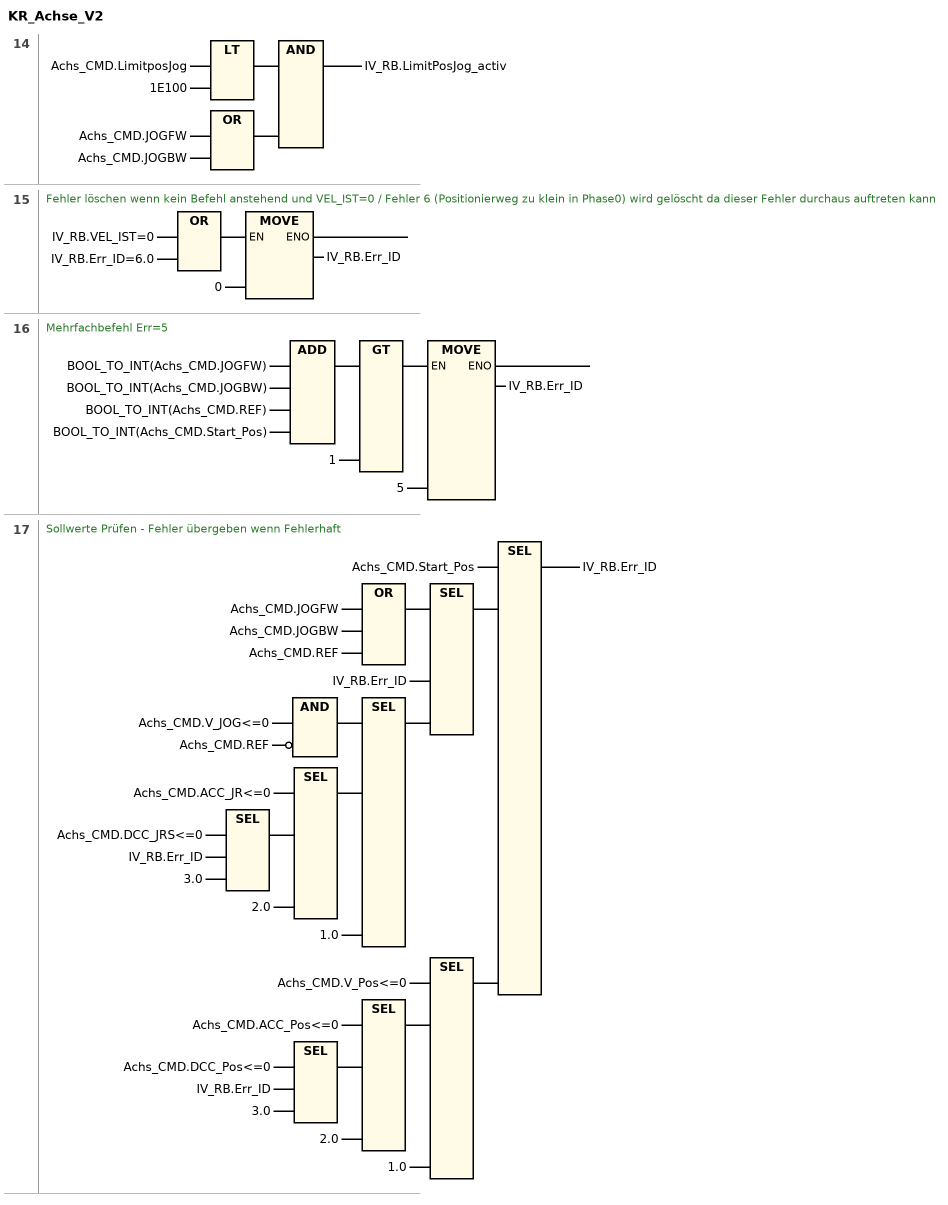
// NETWORK 14
IV_RB.LimitPosJog_activ := Achs_CMD.LimitposJog < 1E100 AND (Achs_CMD.JOGFW OR Achs_CMD.JOGBW);

// NETWORK 15
// Fehler löschen wenn kein Befehl anstehend und VEL_IST=0 / Fehler 6 (Positionierweg zu klein in Phase0) wird gelöscht da dieser Fehler durchaus auftreten kann
IF (IV_RB.VEL_IST=0) OR (IV_RB.Err_ID=6.0) THEN IV_RB.Err_ID := 0; END_IF

// NETWORK 16
// Mehrfachbefehl Err=5
IF (BOOL_TO_INT(Achs_CMD.JOGFW)) + (BOOL_TO_INT(Achs_CMD.JOGBW)) + (BOOL_TO_INT(Achs_CMD.REF)) + (BOOL_TO_INT(Achs_CMD.Start_Pos)) > 1 THEN
    IV_RB.Err_ID := 5;
END_IF

// NETWORK 17
// Sollwerte Prüfen - Fehler übergeben wenn Fehlerhaft
IV_RB.Err_ID := SEL(Achs_CMD.Start_Pos, SEL(Achs_CMD.JOGFW OR Achs_CMD.JOGBW OR Achs_CMD.REF, IV_RB.Err_ID, SEL((Achs_CMD.V_JOG<=0) AND NOT Achs_CMD.REF, SEL(Achs_CMD.ACC_JR<=0, SEL(Achs_CMD.DCC_JRS<=0, IV_RB.Err_ID, 3.0), 2.0), 1.0)), SEL(Achs_CMD.V_Pos<=0, SEL(Achs_CMD.ACC_Pos<=0, SEL(Achs_CMD.DCC_Pos<=0, IV_RB.Err_ID, 3.0), 2.0), 1.0));

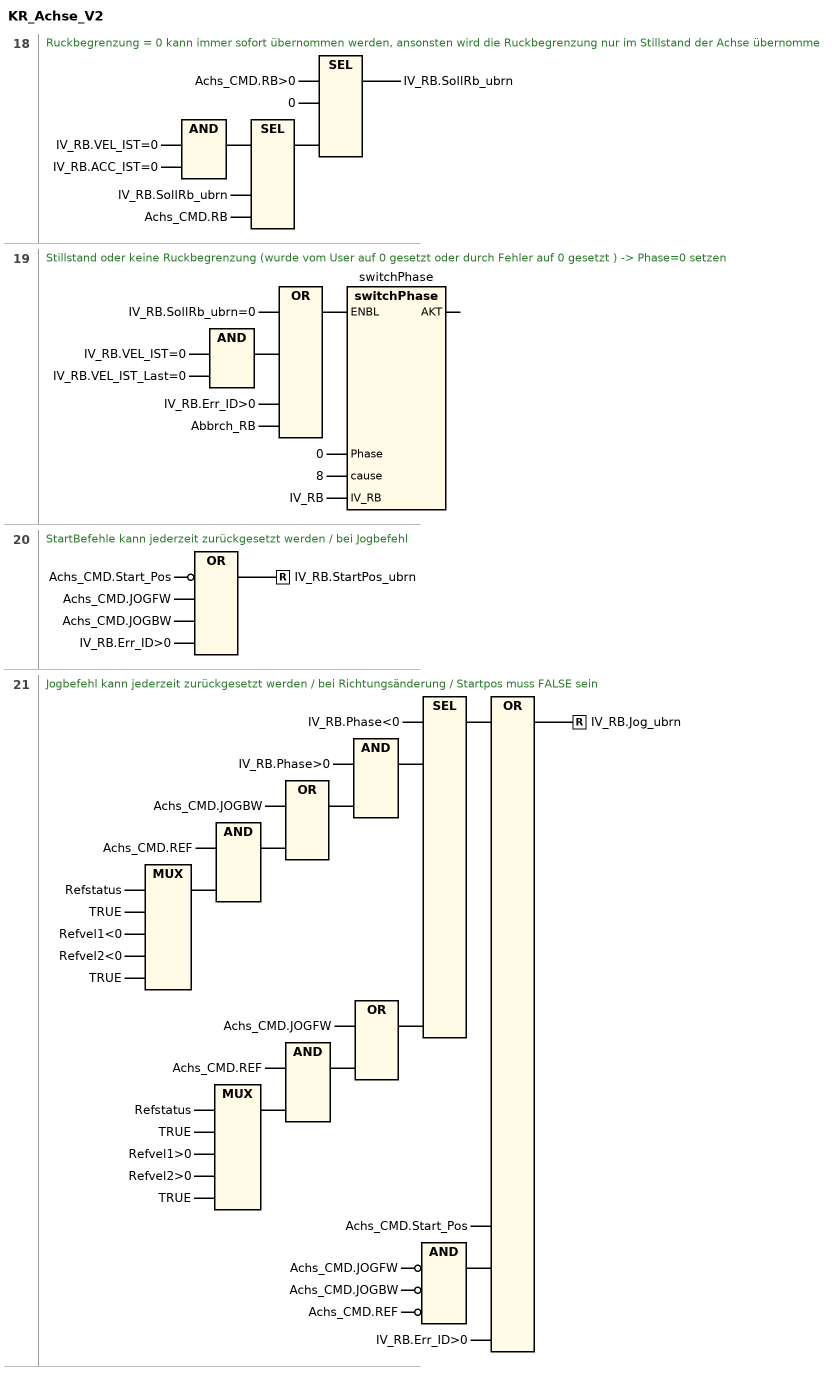
// NETWORK 18
// Ruckbegrenzung = 0 kann immer sofort übernommen werden, ansonsten wird die Ruckbegrenzung nur im Stillstand der Achse übernomme
IV_RB.SollRb_ubrn := SEL(Achs_CMD.RB>0, 0, SEL((IV_RB.VEL_IST=0) AND (IV_RB.ACC_IST=0), IV_RB.SollRb_ubrn, Achs_CMD.RB));

// NETWORK 19
// Stillstand oder keine Ruckbegrenzung (wurde vom User auf 0 gesetzt oder durch Fehler auf 0 gesetzt ) -> Phase=0 setzen
switchPhase(
    ENBL := (IV_RB.SollRb_ubrn=0) OR (IV_RB.VEL_IST=0) AND (IV_RB.VEL_IST_Last=0) OR (IV_RB.Err_ID>0) OR Abbrch_RB,
    Phase := 0,
    cause := 8,
    IV_RB := IV_RB);

// NETWORK 20
// StartBefehle kann jederzeit zurückgesetzt werden / bei Jogbefehl
IV_RB.StartPos_ubrn R= NOT Achs_CMD.Start_Pos OR Achs_CMD.JOGFW OR Achs_CMD.JOGBW OR (IV_RB.Err_ID>0);

// NETWORK 21
// Jogbefehl kann jederzeit zurückgesetzt werden / bei Richtungsänderung / Startpos muss FALSE sein
IV_RB.Jog_ubrn R= SEL(IV_RB.Phase<0, (IV_RB.Phase>0) AND (Achs_CMD.JOGBW OR Achs_CMD.REF AND MUX(Refstatus, TRUE, Refvel1<0, Refvel2<0, TRUE)), Achs_CMD.JOGFW OR Achs_CMD.REF AND MUX(Refstatus, TRUE, Refvel1>0, Refvel2>0, TRUE)) OR Achs_CMD.Start_Pos OR NOT Achs_CMD.JOGFW AND NOT Achs_CMD.JOGBW AND NOT Achs_CMD.REF OR (IV_RB.Err_ID>0);

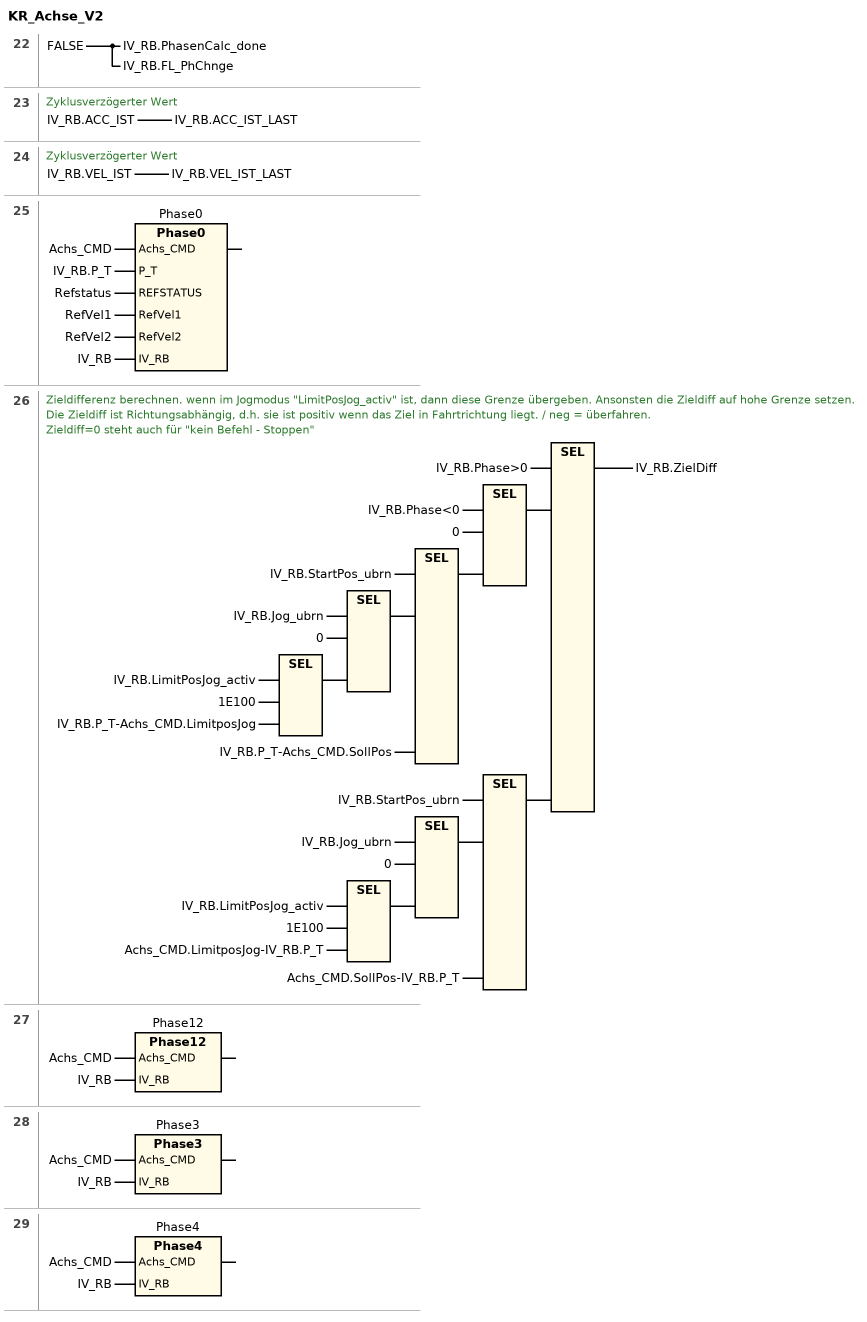
// NETWORK 22
IV_RB.PhasenCalc_done := FALSE;
IV_RB.FL_PhChnge := FALSE;

// NETWORK 23
// Zyklusverzögerter Wert
IV_RB.ACC_IST_LAST := IV_RB.ACC_IST;

// NETWORK 24
// Zyklusverzögerter Wert
IV_RB.VEL_IST_LAST := IV_RB.VEL_IST;

// NETWORK 25
Phase0(
    Achs_CMD := Achs_CMD,
    P_T := IV_RB.P_T,
    REFSTATUS := Refstatus,
    RefVel1 := RefVel1,
    RefVel2 := RefVel2,
    IV_RB := IV_RB);

// NETWORK 26
// 					Zieldifferenz berechnen. wenn im Jogmodus "LimitPosJog_activ" ist, dann diese Grenze übergeben. Ansonsten die Zieldiff auf hohe Grenze setzen.
// Die Zieldiff ist Richtungsabhängig, d.h. sie ist positiv wenn das Ziel in Fahrtrichtung liegt. / neg = überfahren.
// Zieldiff=0 steht auch für "kein Befehl - Stoppen"
//
IV_RB.ZielDiff := SEL(IV_RB.Phase>0, SEL(IV_RB.Phase<0, 0, SEL(IV_RB.StartPos_ubrn, SEL(IV_RB.Jog_ubrn, 0, SEL(IV_RB.LimitPosJog_activ, 1E100, IV_RB.P_T-Achs_CMD.LimitposJog)), IV_RB.P_T-Achs_CMD.SollPos)), SEL(IV_RB.StartPos_ubrn, SEL(IV_RB.Jog_ubrn, 0, SEL(IV_RB.LimitPosJog_activ, 1E100, Achs_CMD.LimitposJog-IV_RB.P_T)), Achs_CMD.SollPos-IV_RB.P_T));

// NETWORK 27
Phase12(Achs_CMD := Achs_CMD, IV_RB := IV_RB);

// NETWORK 28
Phase3(Achs_CMD := Achs_CMD, IV_RB := IV_RB);

// NETWORK 29
Phase4(Achs_CMD := Achs_CMD, IV_RB := IV_RB);

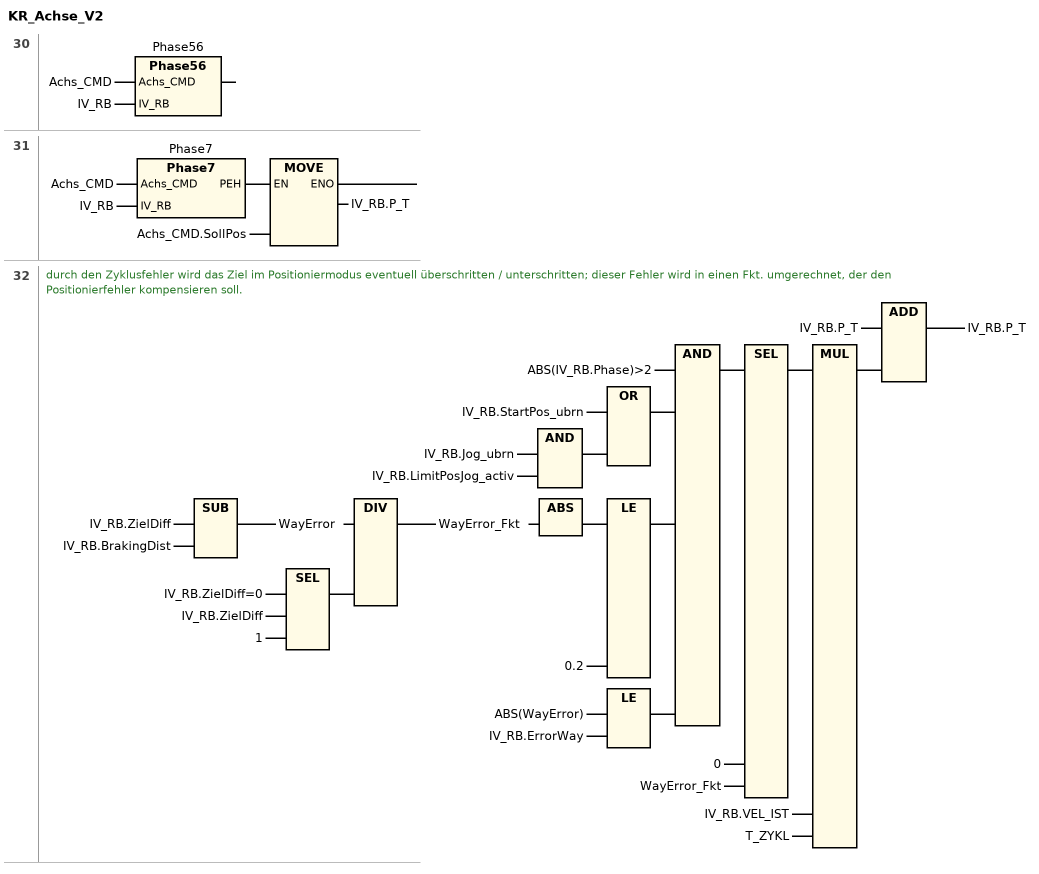
// NETWORK 30
Phase56(Achs_CMD := Achs_CMD, IV_RB := IV_RB);

// NETWORK 31
Phase7(Achs_CMD := Achs_CMD, IV_RB := IV_RB);
IF Phase7.PEH THEN IV_RB.P_T := Achs_CMD.SollPos; END_IF

// NETWORK 32
// durch den Zyklusfehler wird das Ziel im Positioniermodus eventuell überschritten / unterschritten; dieser Fehler wird in einen Fkt. umgerechnet, der den Positionierfehler kompensieren soll.
_w2 := IV_RB.ZielDiff - IV_RB.BrakingDist;
WayError := _w2;
_w3 := _w2 / SEL(IV_RB.ZielDiff=0, IV_RB.ZielDiff, 1);
WayError_Fkt := _w3;
IV_RB.P_T := IV_RB.P_T + SEL((ABS(IV_RB.Phase)>2) AND (IV_RB.StartPos_ubrn OR IV_RB.Jog_ubrn AND IV_RB.LimitPosJog_activ) AND ABS(_w3) <= 0.2 AND (ABS(WayError)) <= IV_RB.ErrorWay, 0, WayError_Fkt) * IV_RB.VEL_IST * T_ZYKL;

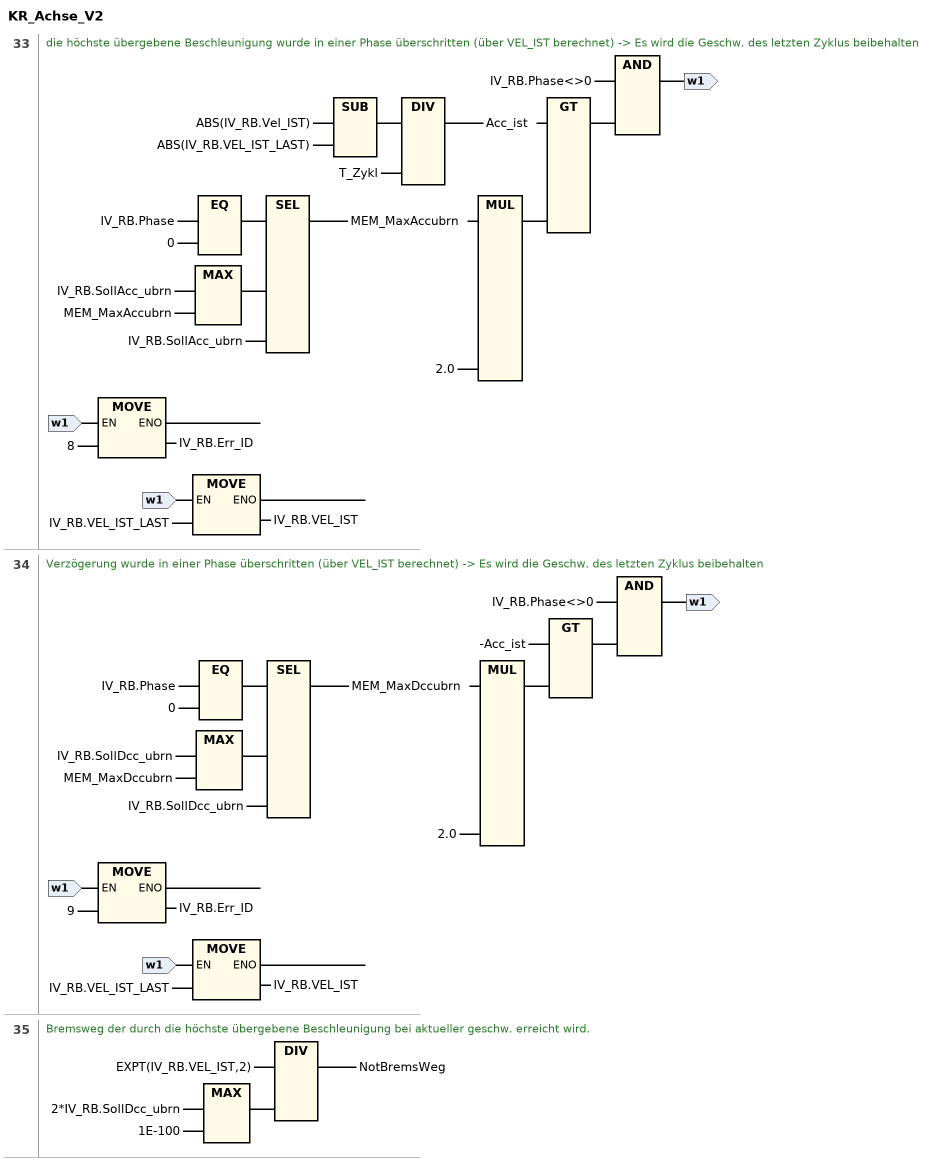
// NETWORK 33
// die höchste übergebene Beschleunigung wurde in einer Phase überschritten (über VEL_IST berechnet) -> Es wird die Geschw. des letzten Zyklus beibehalten
_w4 := ((ABS(IV_RB.Vel_IST)) - (ABS(IV_RB.VEL_IST_LAST))) / T_Zykl;
Acc_ist := _w4;
_w5 := SEL(IV_RB.Phase = 0, MAX(IV_RB.SollAcc_ubrn, MEM_MaxAccubrn), IV_RB.SollAcc_ubrn);
MEM_MaxAccubrn := _w5;
_w6 := (IV_RB.Phase<>0) AND _w4 > _w5 * 2.0;
IF _w6 THEN IV_RB.Err_ID := 8; END_IF
IF _w6 THEN IV_RB.VEL_IST := IV_RB.VEL_IST_LAST; END_IF

// NETWORK 34
// Verzögerung wurde in einer Phase überschritten (über VEL_IST berechnet) -> Es wird die Geschw. des letzten Zyklus beibehalten
_w7 := SEL(IV_RB.Phase = 0, MAX(IV_RB.SollDcc_ubrn, MEM_MaxDccubrn), IV_RB.SollDcc_ubrn);
MEM_MaxDccubrn := _w7;
_w8 := (IV_RB.Phase<>0) AND (-Acc_ist) > _w7 * 2.0;
IF _w8 THEN IV_RB.Err_ID := 9; END_IF
IF _w8 THEN IV_RB.VEL_IST := IV_RB.VEL_IST_LAST; END_IF

// NETWORK 35
// Bremsweg der durch die höchste übergebene Beschleunigung bei aktueller geschw. erreicht wird.
NotBremsWeg := (EXPT(IV_RB.VEL_IST,2)) / MAX(2*IV_RB.SollDcc_ubrn, 1E-100);

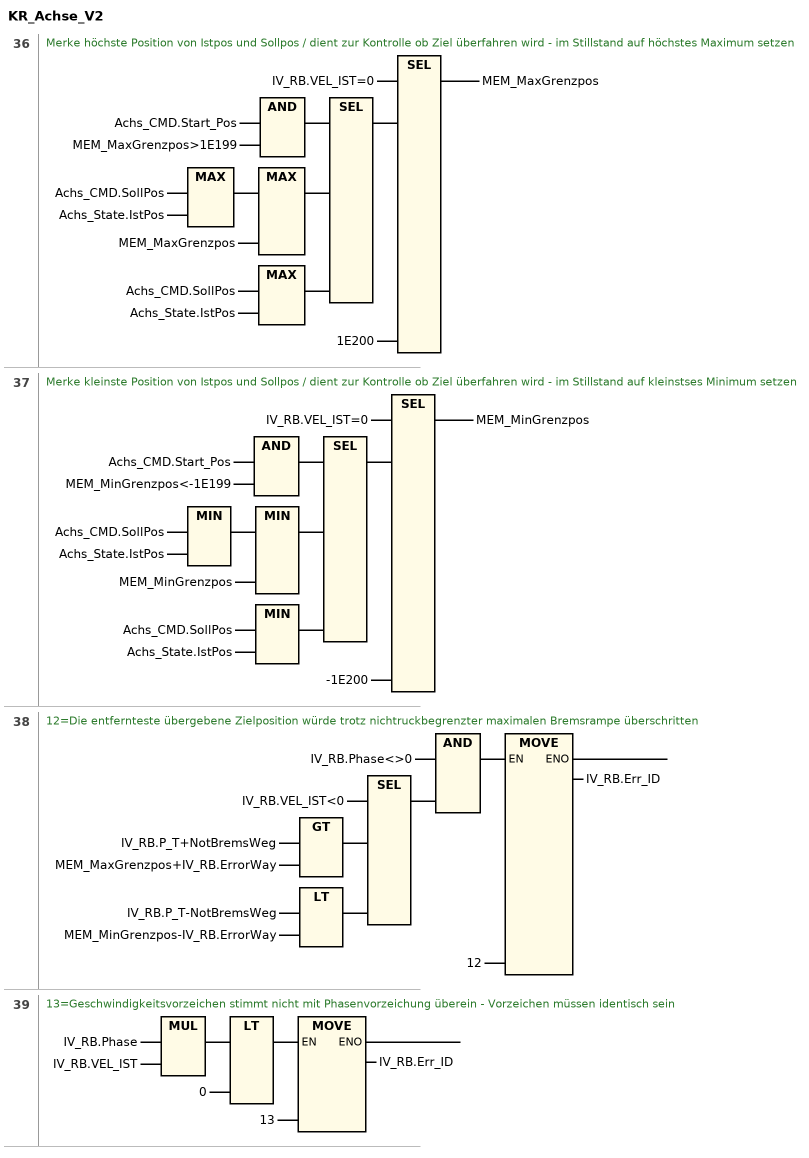
// NETWORK 36
// Merke höchste Position von Istpos und Sollpos / dient zur Kontrolle ob Ziel überfahren wird - im Stillstand auf höchstes Maximum setzen
MEM_MaxGrenzpos := SEL(IV_RB.VEL_IST=0, SEL(Achs_CMD.Start_Pos AND (MEM_MaxGrenzpos>1E199), MAX(MAX(Achs_CMD.SollPos, Achs_State.IstPos), MEM_MaxGrenzpos), MAX(Achs_CMD.SollPos, Achs_State.IstPos)), 1E200);

// NETWORK 37
// Merke kleinste Position von Istpos und Sollpos / dient zur Kontrolle ob Ziel überfahren wird - im Stillstand auf kleinstses Minimum setzen
MEM_MinGrenzpos := SEL(IV_RB.VEL_IST=0, SEL(Achs_CMD.Start_Pos AND (MEM_MinGrenzpos<-1E199), MIN(MIN(Achs_CMD.SollPos, Achs_State.IstPos), MEM_MinGrenzpos), MIN(Achs_CMD.SollPos, Achs_State.IstPos)), -1E200);

// NETWORK 38
// 12=Die entfernteste übergebene Zielposition würde trotz nichtruckbegrenzter maximalen Bremsrampe überschritten
IF (IV_RB.Phase<>0) AND SEL(IV_RB.VEL_IST<0, (IV_RB.P_T+NotBremsWeg) > (MEM_MaxGrenzpos+IV_RB.ErrorWay), (IV_RB.P_T-NotBremsWeg) < (MEM_MinGrenzpos-IV_RB.ErrorWay)) THEN
    IV_RB.Err_ID := 12;
END_IF

// NETWORK 39
// 13=Geschwindigkeitsvorzeichen stimmt nicht mit Phasenvorzeichung überein - Vorzeichen müssen identisch sein
IF IV_RB.Phase * IV_RB.VEL_IST < 0 THEN IV_RB.Err_ID := 13; END_IF

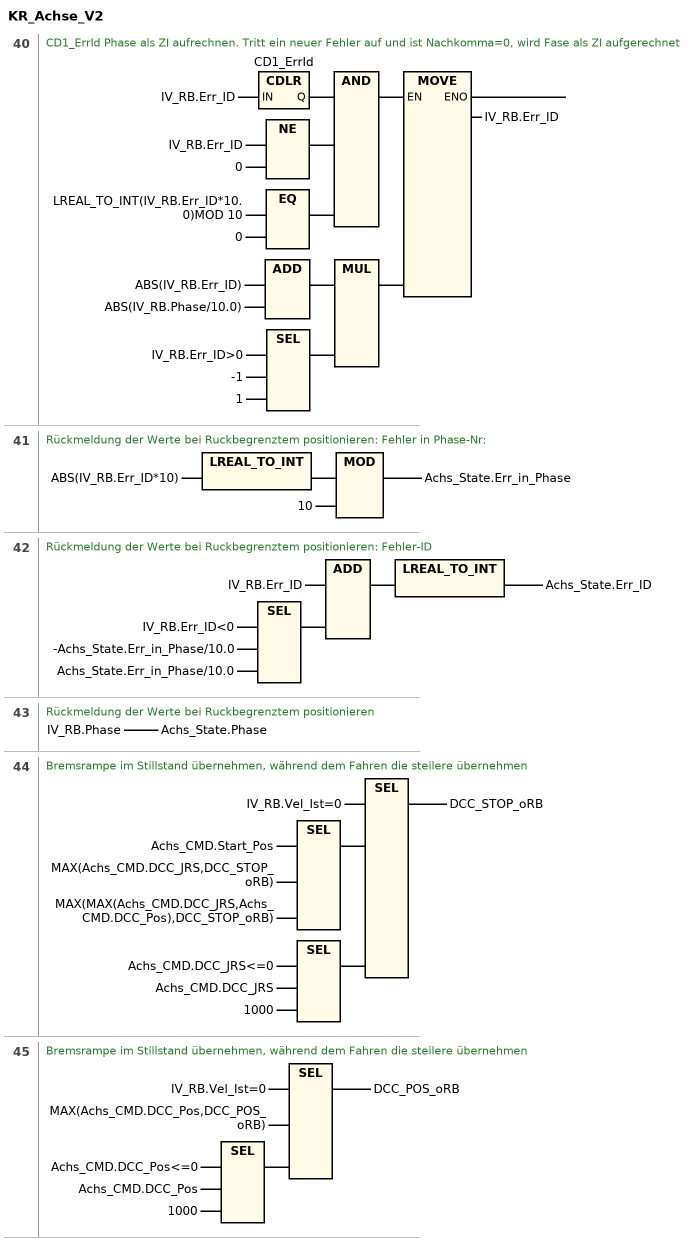
// NETWORK 40
// CD1_ErrId Phase als ZI aufrechnen. Tritt ein neuer Fehler auf und ist Nachkomma=0, wird Fase als ZI aufgerechnet
CD1_ErrId(IN := IV_RB.Err_ID); // CDLR
IF CD1_ErrId.Q AND IV_RB.Err_ID <> 0 AND (LREAL_TO_INT(IV_RB.Err_ID*10.0)MOD 10) = 0 THEN
    IV_RB.Err_ID := ((ABS(IV_RB.Err_ID)) + (ABS(IV_RB.Phase/10.0))) * SEL(IV_RB.Err_ID>0, -1, 1);
END_IF

// NETWORK 41
// Rückmeldung der Werte bei Ruckbegrenztem positionieren: Fehler in Phase-Nr:
Achs_State.Err_in_Phase := LREAL_TO_INT(ABS(IV_RB.Err_ID*10)) MOD 10;

// NETWORK 42
// Rückmeldung der Werte bei Ruckbegrenztem positionieren: Fehler-ID
Achs_State.Err_ID := LREAL_TO_INT(IV_RB.Err_ID + SEL(IV_RB.Err_ID<0, -Achs_State.Err_in_Phase/10.0, Achs_State.Err_in_Phase/10.0));

// NETWORK 43
// Rückmeldung der Werte bei Ruckbegrenztem positionieren
Achs_State.Phase := IV_RB.Phase;

// NETWORK 44
// Bremsrampe im Stillstand übernehmen, während dem Fahren die steilere übernehmen
DCC_STOP_oRB := SEL(IV_RB.Vel_Ist=0, SEL(Achs_CMD.Start_Pos, MAX(Achs_CMD.DCC_JRS,DCC_STOP_oRB), MAX(MAX(Achs_CMD.DCC_JRS,Achs_CMD.DCC_Pos),DCC_STOP_oRB)), SEL(Achs_CMD.DCC_JRS<=0, Achs_CMD.DCC_JRS, 1000));

// NETWORK 45
// Bremsrampe im Stillstand übernehmen, während dem Fahren die steilere übernehmen
DCC_POS_oRB := SEL(IV_RB.Vel_Ist=0, MAX(Achs_CMD.DCC_Pos,DCC_POS_oRB), SEL(Achs_CMD.DCC_Pos<=0, Achs_CMD.DCC_Pos, 1000));

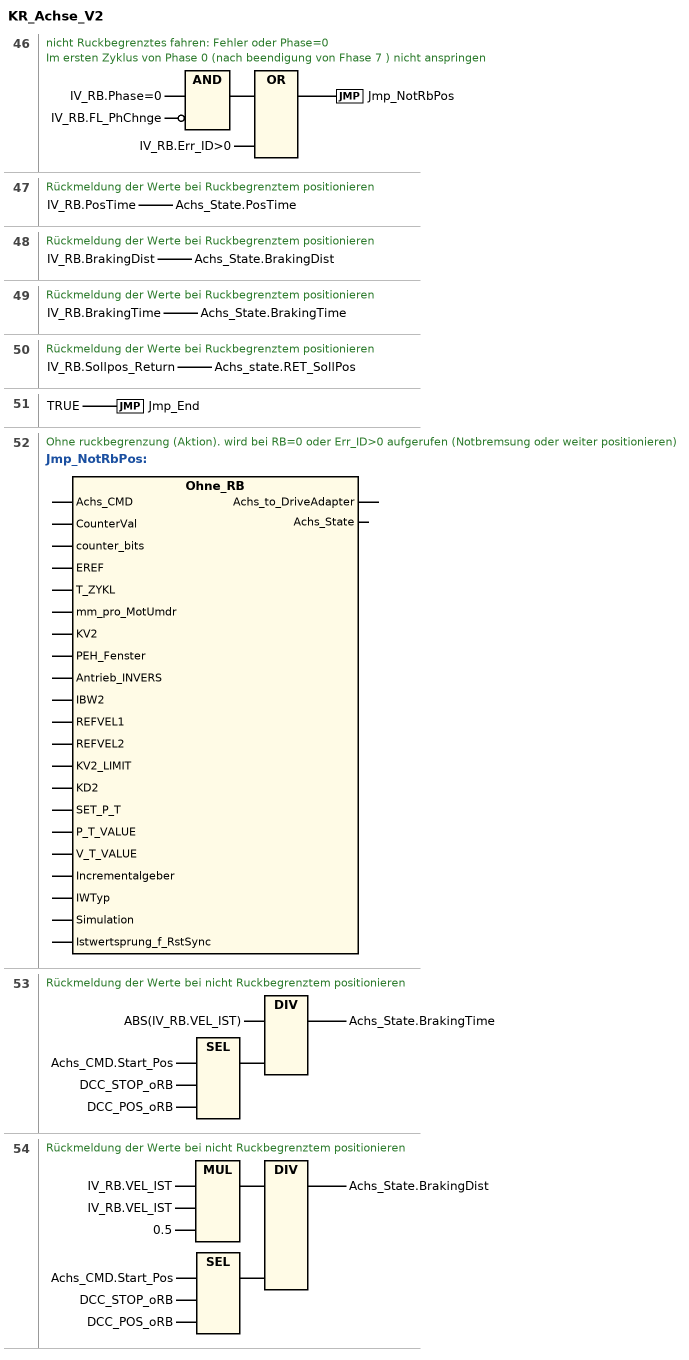
// NETWORK 46
// 					nicht Ruckbegrenztes fahren: Fehler oder Phase=0
// Im ersten Zyklus von Phase 0 (nach beendigung von Fhase 7 ) nicht anspringen
//
IF (IV_RB.Phase=0) AND NOT IV_RB.FL_PhChnge OR (IV_RB.Err_ID>0) THEN JMP Jmp_NotRbPos; END_IF

// NETWORK 47
// Rückmeldung der Werte bei Ruckbegrenztem positionieren
Achs_State.PosTime := IV_RB.PosTime;

// NETWORK 48
// Rückmeldung der Werte bei Ruckbegrenztem positionieren
Achs_State.BrakingDist := IV_RB.BrakingDist;

// NETWORK 49
// Rückmeldung der Werte bei Ruckbegrenztem positionieren
Achs_State.BrakingTime := IV_RB.BrakingTime;

// NETWORK 50
// Rückmeldung der Werte bei Ruckbegrenztem positionieren
Achs_state.RET_SollPos := IV_RB.Sollpos_Return;

// NETWORK 51
JMP Jmp_End;

// NETWORK 52
// Ohne ruckbegrenzung (Aktion). wird bei RB=0 oder Err_ID>0 aufgerufen (Notbremsung oder weiter positionieren)
Jmp_NotRbPos:
Ohne_RB();

// NETWORK 53
// Rückmeldung der Werte bei nicht Ruckbegrenztem positionieren
Achs_State.BrakingTime := (ABS(IV_RB.VEL_IST)) / SEL(Achs_CMD.Start_Pos, DCC_STOP_oRB, DCC_POS_oRB);

// NETWORK 54
// Rückmeldung der Werte bei nicht Ruckbegrenztem positionieren
Achs_State.BrakingDist := (IV_RB.VEL_IST * IV_RB.VEL_IST * 0.5) / SEL(Achs_CMD.Start_Pos, DCC_STOP_oRB, DCC_POS_oRB);

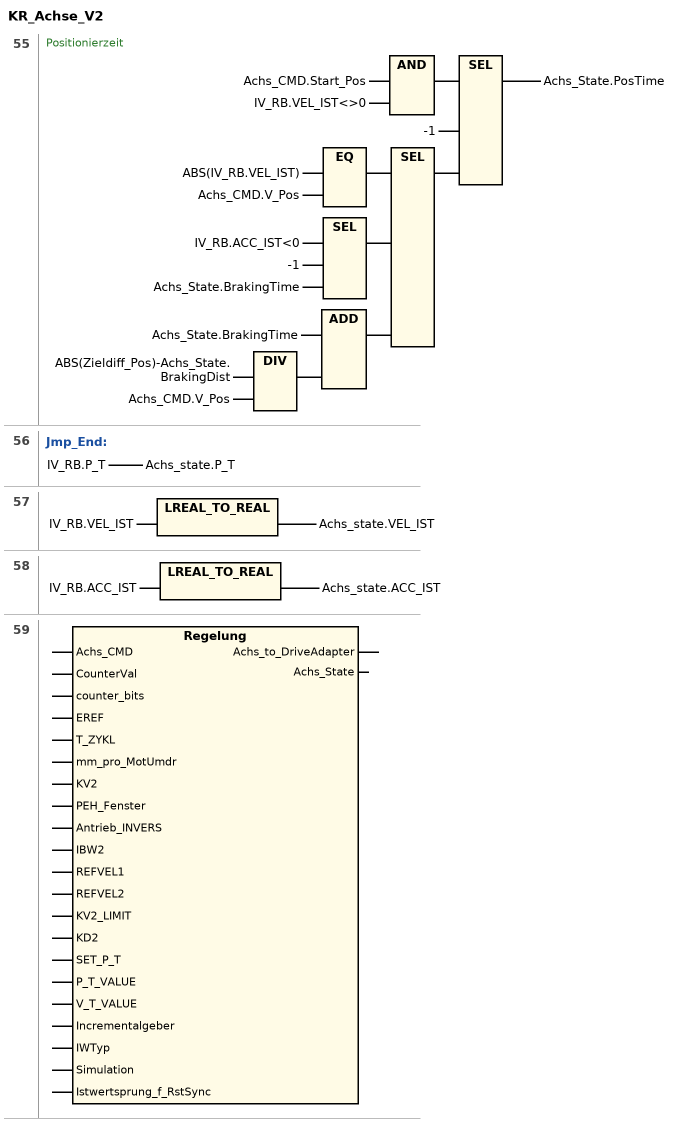
// NETWORK 55
// Positionierzeit
Achs_State.PosTime := SEL(Achs_CMD.Start_Pos AND (IV_RB.VEL_IST<>0), -1, SEL((ABS(IV_RB.VEL_IST)) = Achs_CMD.V_Pos, SEL(IV_RB.ACC_IST<0, -1, Achs_State.BrakingTime), Achs_State.BrakingTime + (ABS(Zieldiff_Pos)-Achs_State.BrakingDist) / Achs_CMD.V_Pos));

// NETWORK 56
Jmp_End:
Achs_state.P_T := IV_RB.P_T;

// NETWORK 57
Achs_state.VEL_IST := LREAL_TO_REAL(IV_RB.VEL_IST);

// NETWORK 58
Achs_state.ACC_IST := LREAL_TO_REAL(IV_RB.ACC_IST);

// NETWORK 59
Regelung();

ACTION encoder:
(*  ##################### Aktion: Umrechnung Incremente in Istwert  ############################### *)

(*##################### S I M U L A T I O N ###################*)
IF Simulation THEN
	Sim_EncoderVal:=Achs_to_DriveAdapter.motorSpeed/60.0*T_ZYKL*mm_pro_MotUmdr/IBW2+Sim_EncoderVal;
	IF Sim_EncoderVal>2147483647 THEN Sim_EncoderVal:=Sim_EncoderVal-2147483647;
	ELSIF Sim_EncoderVal<-2147483647 THEN Sim_EncoderVal:=Sim_EncoderVal+2147483647;
	END_IF
	CounterVal :=LREAL_TO_DINT(Sim_EncoderVal);
	counter_bits := MIN(counter_bits,31);
END_IF
(* ############ Ende SIMULATION #############################*)

EmptyBits:=(32-counter_bits);
EncBitMask:=SHR(16#FFFF_FFFF,EmptyBits); (*Bitmaske aller verwendeten Encoder-Bits *)
CountLimit1:=EncBitMask/4;(* wird für Counter-Überschlagsberechnung benutzt*)
CountLimit2:=CountLimit1*3;(* wird für Counter-Überschlagsberechnung benutzt*)

IF Incrementalgeber THEN
	IF Antrieb_invers THEN
		copy_Counter:=DINT_TO_DWORD(-CounterVal) AND EncBitMask;(*nicht verwendete Bits ausblenden ( zur Sicherheit wenn obere Bits des encoders trotzdem Signale liefern) *)
	ELSE
		copy_Counter:=DINT_TO_DWORD(CounterVal) AND EncBitMask;(*nicht verwendete Bits ausblenden ( zur Sicherheit wenn obere Bits des encoders trotzdem Signale liefern) *)
	END_IF

	IF copy_Counter < CountLimit1 AND copy_Counter_Last > CountLimit2 THEN Incr_Offset:=Incr_Offset+DWORD_TO_LREAL(EncBitMask)+1.0; (*Überschlag vorwärts*)
	ELSIF copy_Counter > CountLimit2 AND copy_Counter_Last < CountLimit1 THEN Incr_Offset:=Incr_Offset-DWORD_TO_LREAL(EncBitMask)-1.0;(*Überschlag rückärts*)
	END_IF

	TempDint1:=DWORD_TO_DINT(SHL(copy_Counter,EmptyBits));
	TempDint2:=DWORD_TO_DINT(SHL(copy_Counter_Last,EmptyBits));
	TempDint1:=ABS(TempDint1-TempDint2);
	TempDint1:=SHR(TempDint1,EmptyBits);
	IF TempDint1*IBW2 > Istwertsprung_f_RstSync THEN Achs_State.SYNC:=FALSE;END_IF

ELSE (*Absolutachse*)

	(*Der IWT wird so berechnet, daß durch Summe mit dem CounterVal ein Wert entsteht, der beim typischen Achsen-Istwert "IWT" genau der Hälfte vom Vollen Counter-Val entspricht, dadurch wir der Zählerüberschlag in pos. und neg. Richtung in gleicher Entfernung gesetzt*)
	(*Bits die den Wertebereich eines 32bit Datentyps übschreiten werden eliminiert.*)
	IWT_Offset:=LINT_TO_DINT(LREAL_TO_LINT((Achs_CMD.IstWertOffset-IWTyp)/(IBW2) +DWORD_TO_LREAL(EncBitMask/2)) MOD 16#1_0000_0000);
 	IF Antrieb_INVERS THEN
  		copy_Counter:= DINT_TO_DWORD((-CounterVal)+IWT_Offset);
 	ELSE
  		copy_Counter:=DINT_TO_DWORD(CounterVal+IWT_Offset);
	END_IF
	copy_Counter:=copy_Counter AND EncBitMask;

	IF copy_Counter < CountLimit1 AND copy_Counter_Last > CountLimit2 THEN Set_PT_Eq_Istpos:=TRUE; (*Überschlag vorwärts*)
	ELSIF copy_Counter > CountLimit2 AND copy_Counter_Last < CountLimit1 THEN Set_PT_Eq_Istpos:=TRUE;(*Überschlag rückärts*)
	END_IF

END_IF
copy_Counter_Last:=copy_Counter;


(*############# Referenzmodus: ohne Nullspur oder mit Nullspur ( mit EL,LV COUNTER) #############*)
IF Achs_CMD.REF AND Incrementalgeber THEN (*0=Referenz ohne Nullspur*)
	IF REFSTATUS=0 THEN (*Referenzfahrt hat noch nicht begonnen*)
		Achs_State.SYNC:=FALSE;(*Achs_State.SYNC löschen bei Anwahl von Ref-Modus*)
		IF NOT EREF THEN REFSTATUS:=1; (*Refstatus: suche Endschalter*)
		ELSE REFSTATUS:=2; (*Refstatus: Endschalter belegt, suche negative Flanke Endschalter*)
		END_IF
	ELSIF REFSTATUS=1 AND EREF THEN REFSTATUS:=2; (*Wenn Status=suche Endschalter und EREF belegt, dann Status=2*)
	ELSIF REFSTATUS=2 AND NOT EREF THEN

		IF (REFVEL2 * Achs_State.Vel_Ist) < 0 THEN (*Flanke Endschalter ist aufgetreten, aber die Sollrichtung und die Fahrrichtung stimmen nicht überein: Referenzfahrt neu beginnen*)
			REFSTATUS:=0;
		ELSE
			REFSTATUS:=7; (*negative Flanke Endschalter: Refstatus=7 (fertig, Istwert neu setzen*)
			Incr_Offset:=Achs_CMD.RefPos/IBW2-DWORD_TO_LREAL(copy_Counter);Achs_State.SYNC:=TRUE;Set_PT_Eq_Istpos:=TRUE;
		END_IF
	END_IF


ELSE REFSTATUS:=0;(*Wenn nicht REF-Modus, dann REFSTATUS=0*)

END_IF

(*Istposition setzen*)
IF Achs_CMD.SETPOS AND Incrementalgeber THEN
	Incr_Offset:=Achs_CMD.RefPos/IBW2-DWORD_TO_LREAL(copy_Counter);Set_PT_Eq_Istpos:=TRUE;Achs_State.SYNC:=TRUE;
END_IF

IF Achs_CMD.IstWertOffset <> IstWertOffset_LAST THEN Set_PT_Eq_Istpos:=TRUE;END_IF
IstWertOffset_LAST:=Achs_CMD.IstWertOffset;

(* Ermittlung des Geberistwertes *)

IF Incrementalgeber THEN
	Achs_State.IstPos:=(copy_Counter+Incr_Offset)*IBW2+Achs_CMD.IstWertOffset;(*Incrementalgeber: Der Achs_CMD.IstWertOffset wird dierekt dem Istwert aufgerechnet*)
ELSE
	Achs_State.IstPos:=DWORD_TO_LREAL(copy_Counter)*IBW2 - DWORD_TO_LREAL(EncBitMask/2)*IBW2+IWTyp;(*Absolutachse: Der Achs_CMD.IstWertOffset ist bereits den Incrementwert aufgerechnet, der halbe Gesamtincrement-Bereich und der Typ.Istwert, die ebenfalls aufgerechnet wurden, müss hier wieder abgerechnet werden: 536870912.0 D = 16#8000_0000 H*)
END_IF
END_ACTION

ACTION ohne_RB:
(*## Achsen-Steuerung, Online Positionsänderung bei Ruckbegrenztem positionieren, Ruckbegrenztes abbremsen bei wegnahme von Start  ###*)
(*###########################################################################################################*)
IF Achs_CMD.ACC_JR<=0 THEN Achs_CMD.ACC_JR:=1;END_IF
Bremsweg_Jog:=IV_RB.VEL_IST*IV_RB.VEL_IST/(2*DCC_STOP_oRB);

(*################################ REFERENZFAHRT ################################################*)
IF IV_RB.Err_ID=0 AND Achs_CMD.REF AND NOT Achs_State.Sync THEN
	IF REFSTATUS=1 THEN V_SOLL:=REFVEL1;
	ELSE V_SOLL:=REFVEL2;
	END_IF
	IF V_SOLL>0 THEN (*Fahrgeschwindigkeit grösser 0 *)
		IF IV_RB.Vel_Ist >= 0 THEN (*Achse steht oder fährt vor*)
			IF IV_RB.Vel_Ist > V_SOLL THEN (*Achse muß abbremsen, da Soll-Vel aufgrund DECC bereits kleiner als aktuelle IV_RB.Vel_Ist ist*)
				IV_RB.Vel_Ist:=MAX(V_SOLL,(IV_RB.Vel_Ist-Achs_CMD.DCC_JRS*T_ZYKL)); (*Geschwindigkeit verringern, Staus: DEC,vorwärts*)
			ELSIF IV_RB.Vel_Ist < V_SOLL THEN (*Achse muß beschleunigen, da V_Soll noch nicht erreicht ist*)
				IV_RB.Vel_Ist:=MIN(V_Soll,(IV_RB.Vel_Ist+Achs_CMD.ACC_JR*T_ZYKL)); (*Geschwindigkeit erhöhen, STATUS=ACC,vorwärts*)
			END_IF
		ELSE (*Achse fährt zurück, JOG Vor verlangt: abbremsen auf 0 *)
			IV_RB.Vel_Ist:=IV_RB.Vel_Ist+Achs_CMD.DCC_JRS*T_ZYKL;
		END_IF
			IV_RB.P_T:=IV_RB.P_T+IV_RB.Vel_Ist*T_ZYKL;
	ELSE (*Fahrgeschwindigkeit kleiner 0*)
		IF IV_RB.Vel_Ist <= 0 THEN (*Achse steht oder fährt zurück*)
			IF IV_RB.Vel_Ist < V_SOLL THEN (*Achse muß abbremsen, da Soll-Vel aufgrund DECC bereits kleiner als aktuelle IV_RB.Vel_Ist ist*)
				IV_RB.Vel_Ist:=MIN(V_SOLL,(IV_RB.Vel_Ist+Achs_CMD.DCC_JRS*T_ZYKL)); (*Geschwindigkeit verringern, Staus: DEC,rückwärts*)
			ELSIF IV_RB.Vel_Ist > V_SOLL THEN (*Achse muß beschleunigen, da V_Soll noch nicht erreicht ist*)
				IV_RB.Vel_Ist:=MAX(V_Soll,(IV_RB.Vel_Ist-Achs_CMD.ACC_JR*T_ZYKL)); (*Geschwindigkeit erhöhen, STATUS=ACC,rückwärts*)
			END_IF
		ELSE (*Achse fährt vor, JOG zur verlangt: abbremsen auf 0 *)
			IV_RB.Vel_Ist:=IV_RB.Vel_Ist-Achs_CMD.DCC_JRS*T_ZYKL;
		END_IF
			IV_RB.P_T:=IV_RB.P_T+IV_RB.Vel_Ist*T_ZYKL;
	END_IF
(*########################## Positionieren OHNE Ruckbegrenzung ######################################*)
(*POSITIONIEREN POSITIONIEREN POSITIONIEREN POSITIONIEREN POSITIONIEREN POSITIONIEREN POSITIONIEREN POSITIONIEREN *)
ELSIF IV_RB.Err_ID<=0 AND (Achs_CMD.Start_Pos OR (Achs_CMD.REF AND Achs_State.Sync)) THEN (*Wenn Positioniermodus ohne Ruckbegrenzung ODER Wenn REF-Modus UND SNYC gesetzt, dann Positionieren *)
 	IF Achs_CMD.Start_Pos THEN (*Wenn Positioiermodus, dann ist Sollposition=Sollpos*)
		Sollpos:=Achs_CMD.Sollpos;V_POS:=MAX(0,Achs_CMD.V_POS);
		ACC_POS:=ABS(Achs_CMD.ACC_POS);
		Zieldiff_Pos:=SollPos-IV_RB.P_T; (* Differenz zum Ziel= Zielposition - Theoretischer Echtzeit-Position*)
		IF ABS((IV_RB.Vel_Ist*IV_RB.Vel_Ist)/(2*Achs_CMD.DCC_POS))<=ABS(Zieldiff_Pos) AND (IV_RB.Vel_Ist*Zieldiff_Pos)>=0 THEN (*Ziel wird durch flachere Rampe nicht überfahren, Rampe übernehmen*)
			DCC_POS_oRB:=ABS(Achs_CMD.DCC_POS);DCC_STOP_oRB:=MAX(Achs_CMD.DCC_JRS,DCC_POS_oRB); (*Beschleunigung nur übernehmen, wenn Ziel dadurch nicht überfahren wird, Vel und Zieldiff müssen selbes Vorzeichen haben*)
		END_IF
	ELSE (*Ansonsten auf Nullpunkt Positionieren (nach REF-Fahrt*)
  		Sollpos:=Achs_CMD.RefPos+Achs_CMD.IstWertOffset;V_POS:=ABS(REFVEL2);ACC_POS:=Achs_CMD.ACC_JR;DCC_POS_oRB:=Achs_CMD.DCC_JRS;
		Zieldiff_Pos:=SollPos-IV_RB.P_T; (* Differenz zum Ziel= Zielposition - Theoretischer Echtzeit-Position*)
	END_IF
	Achs_State.RET_SollPos:=Sollpos;
	PEH_Val:=0.5*DCC_POS_oRB*T_ZYKL*T_ZYKL;PEV_Val:=DCC_POS_oRB*T_ZYKL;
	IF ABS(Zieldiff_Pos)>PEH_Val OR ABS(IV_RB.Vel_Ist)>PEV_Val THEN (*Wenn die Differenz zum Ziel > PEH-Fenster oder IV_RB.Vel_Ist>Geschw.-Diff pro Zyklus aufgrund verzögerungsrampe, dann positionieren*)
		IF Zieldiff_Pos>0 THEN (*Ziel ist in positiver richtung*)
			V_SOLL:=MIN(V_Pos,(SQRT(2*Zieldiff_Pos*DCC_POS_oRB)-0.5*DCC_POS_oRB*T_ZYKL));(*Sollgeschwindigkeit aufgrund Verzögerungssrampe und Restweg*)
			IF IV_RB.Vel_Ist >= 0 THEN (*Achse steht oder fährt vor*)
				IF IV_RB.Vel_Ist > V_SOLL THEN (*Achse muß abbremsen, da Soll-Vel aufgrund DECC bereits kleiner als aktuelle IV_RB.Vel_Ist ist*)
					IV_RB.Vel_Ist:=MAX(V_SOLL,(IV_RB.Vel_Ist-DCC_POS_oRB*T_ZYKL)); (*Geschwindigkeit verringern, Staus: DEC,vorwärts*)
				ELSIF IV_RB.Vel_Ist < V_POS THEN (*Achse muß beschleunigen, da V_Pos noch nicht erreicht ist*)
					IV_RB.Vel_Ist:=MIN(MIN(V_POS,(IV_RB.Vel_Ist+ACC_Pos*T_ZYKL)),V_SOLL);  (*Geschwindigkeit erhöhen, STATUS=ACC,vorwärts*)
				END_IF
			ELSE (*Achse fährt zurück, Ziel ist vorne: umdrehen: auf 0 mit DECC-Rampe*)
				IV_RB.Vel_Ist:=IV_RB.Vel_Ist+DCC_POS_oRB*T_ZYKL; (*abbremsen um zu wenden*)
			END_IF
		ELSE (*Ziel ist in negativer Richtung*)
			V_SOLL:=MAX(-V_Pos,-(SQRT(-2*Zieldiff_Pos*DCC_POS_oRB)-0.5*DCC_POS_oRB*T_ZYKL));(*Sollgeschwindigkeit aufgrund Verzögerungssrampe*)
			IF IV_RB.Vel_Ist <= 0 THEN (*Achse steht oder fährt zurück*)
				IF IV_RB.Vel_Ist < V_SOLL THEN (*Achse muß abbremsen, da Soll-Vel aufgrund DECC bereits positiver als aktuelle IV_RB.Vel_Ist ist*)
					IV_RB.Vel_Ist:=MIN((V_SOLL),(IV_RB.Vel_Ist+DCC_POS_oRB*T_ZYKL));  (*Geschwindigkeit verringern, Staus: DEC,rückwärts*)
				ELSIF IV_RB.Vel_Ist > -V_POS THEN (*Achse muß beschleunigen, da V_Pos noch nicht erreicht ist*)
					IV_RB.Vel_Ist:=MAX(MAX(-V_POS,(IV_RB.Vel_Ist-ACC_Pos*T_ZYKL)),V_SOLL);  (*Geschwindigkeitsbetrag erhöhen, STATUS=ACC,rückwärts*)
				END_IF
			ELSE (*Achse fährt vor, Ziel ist hinten:umdrehen: auf 0 mit DECC*)
				IV_RB.Vel_Ist:=IV_RB.Vel_Ist-DCC_POS_oRB*T_ZYKL;
			END_IF
		END_IF
		IV_RB.P_T:=IV_RB.P_T+IV_RB.Vel_Ist*T_ZYKL; (*Berechnung der Echtzeit-Position*)
	ELSE (*Ziel ist aufgrund PEH und Geschwindigkeit erreicht: Lageregelung aufnehmen*)
		IV_RB.Vel_Ist:=0;
		IV_RB.P_T:=Sollpos;
	END_IF
	(*################### JOG-Betrieb mit konstanter Geschwindigkeit ohne Startrampe ###################*)
(* JOG JOG JOG JOG JOG JOG JOG JOG JOG JOG JOG JOG JOG JOG JOG JOG JOG JOG JOG JOG JOG JOG JOG JOG JOG JOG JOG *)
ELSIF Achs_CMD.JOGFW AND NOT (IV_RB.LimitPosJog_activ AND IV_RB.P_T>(Achs_CMD.LimitposJog-Bremsweg_Jog)) THEN
	V_SOLL:=Achs_CMD.V_JOG;
	IF IV_RB.Vel_Ist >= 0 THEN (*Achse steht oder fährt vor*)
		IF IV_RB.Vel_Ist > V_SOLL THEN (*Achse muß abbremsen, da Soll-Vel aufgrund DECC bereits kleiner als aktuelle IV_RB.Vel_Ist ist*)
			IV_RB.Vel_Ist:=MAX(V_SOLL,(IV_RB.Vel_Ist-DCC_STOP_oRB*T_ZYKL)); (*Geschwindigkeit verringern, Staus: DEC,vorwärts*)
		ELSIF IV_RB.Vel_Ist < V_SOLL THEN (*Achse muß beschleunigen, da V_Soll noch nicht erreicht ist*)
			IV_RB.Vel_Ist:=MIN(V_Soll,(IV_RB.Vel_Ist+Achs_CMD.ACC_JR*T_ZYKL)); (*Geschwindigkeit erhöhen, STATUS=ACC,vorwärts*)
		END_IF
	ELSE (*Achse fährt zurück, JOG Vor verlangt: abbremsen auf 0 *)
		IV_RB.Vel_Ist:=IV_RB.Vel_Ist+DCC_STOP_oRB*T_ZYKL;
	END_IF
	IV_RB.P_T:=IV_RB.P_T+IV_RB.Vel_Ist*T_ZYKL;
ELSIF Achs_CMD.JOGBW AND NOT (IV_RB.LimitPosJog_activ AND IV_RB.P_T<(Achs_CMD.LimitposJog+Bremsweg_Jog)) THEN
	V_SOLL:=-Achs_CMD.V_JOG;
	IF IV_RB.Vel_Ist <= 0 THEN (*Achse steht oder fährt zurück*)
		IF IV_RB.Vel_Ist < V_SOLL THEN (*Achse muß abbremsen, da Soll-Vel aufgrund DECC bereits kleiner als aktuelle IV_RB.Vel_Ist ist*)
			IV_RB.Vel_Ist:=MIN(-V_SOLL,(IV_RB.Vel_Ist+DCC_STOP_oRB*T_ZYKL)); (*Geschwindigkeit verringern, Staus: DEC,rückwärts*)
		ELSIF IV_RB.Vel_Ist > V_SOLL THEN (*Achse muß beschleunigen, da V_Soll noch nicht erreicht ist*)
			IV_RB.Vel_Ist:=MAX(V_Soll,(IV_RB.Vel_Ist-Achs_CMD.ACC_JR*T_ZYKL)); (*Geschwindigkeit erhöhen, STATUS=ACC,rückwärts*)
		END_IF
	ELSE (*Achse fährt vor, JOG zur verlangt: abbremsen auf 0 *)
		IV_RB.Vel_Ist:=IV_RB.Vel_Ist-DCC_STOP_oRB*T_ZYKL;
	END_IF
		IV_RB.P_T:=IV_RB.P_T+IV_RB.Vel_Ist*T_ZYKL;

(*################# Direkte P_T-Vorgabe, z.B. zum zeichnen eines Kreise (PLOTTER) bei dem beide Achsen über Zeitraster gekoppelt sind ###########################*)
ELSIF SET_P_T THEN
	IV_RB.Vel_Ist:=V_T_VALUE; (*Übergabe der Geschwindigkeit*)
	IV_RB.P_T:=P_T_VALUE;
	(*####################### Anhalten, keine Bedingung erfüllt##########################################*)
(* HALT HALT HALT HALT HALT HALT HALT HALT HALT HALT HALT HALT HALT HALT HALT HALT HALT HALT HALT HALT HALT HALT *)
ELSE
	IF ABS(IV_RB.Vel_Ist) > (DCC_STOP_oRB*T_ZYKL) THEN (*Wenn aktuelle Geschw. grösser als Geschwindigkeitsänderung pro Zyklus ist, dann positionieren:*)
		IF  IV_RB.Vel_Ist > 0 THEN (*Bremsen von positiv auf 0, aktuelle Geschw. grösser 0*)
			V_SOLL:=IV_RB.Vel_Ist-DCC_STOP_oRB*T_ZYKL; (* Soll- Geschwindigkeit aufgrund der Bremsrampe*)
			IV_RB.Vel_Ist:=MAX(0,V_SOLL); (* Limitieren auf 0, soll ja stehen bleiben und nicht rückwärts fahren*)
		ELSE
			V_SOLL:=IV_RB.Vel_Ist+DCC_STOP_oRB*T_ZYKL; (* Die neue Geschwindigkeit aufgrund der Bremsrampe*)
			IV_RB.Vel_Ist:=MIN(0,V_SOLL); (* Limitieren auf 0, soll ja stehen bleiben und nicht vorwärts fahren*)
		END_IF
	ELSE
		IV_RB.Vel_Ist:=0;(* Stillstandsgeschw. unterschritten, Lageregelung durch IV_RB.Vel_Ist=0 machen*)
	END_IF
	IV_RB.P_T:=IV_RB.P_T+IV_RB.Vel_Ist*T_ZYKL; (*Die neue Sollposition aufgrund aktueller Geschwindigkeit*)
END_IF

IV_RB.Acc_Ist:=(ABS(IV_RB.Vel_Ist)-ABS(IV_RB.Vel_Ist_LAST))/T_ZYKL;(* Die Ist-Beschleunigung wird bei nichtruckbegrenztem pos. gemessen, positiv bedeutet Beschleunigen, negativ = bremsen*)
END_ACTION

ACTION Regelung:
(*########## Berechnung des Sollwertes aufgrund aktueller Geschwindigkeit UND Schleppabstand*KV-Faktor###############*)

(* Rückmeldungen / Ausgangsvariablen übergeben*)
Achs_State.Schleppabst:=LREAL_TO_REAL(Achs_State.P_T-Achs_State.IstPos);

IF Achs_State.Vel_Ist=0 AND ((Achs_CMD.Start_Pos AND
ABS(Achs_CMD.Sollpos-Achs_State.IstPos)<=PEH_Fenster) OR (Achs_CMD.REF AND  Achs_State.SYNC AND ABS(Achs_CMD.RefPOS-Achs_State.Istpos+Achs_CMD.IstWertOffset)<=PEH_Fenster)) THEN
	Achs_State.PEH:=TRUE;
	Achs_State.RET_SollPos:=Achs_CMD.Sollpos; (*Beim (Ruckbegrenzten) Positionieren wird die Positionier-Routine nicht bearbeitet, wenn Sollpos=Istpos ist, wodurch RET_Sollpos nicht zurückgemeldet wird. Deswegen muss hier explizit nochmals die RET_Sollpos beschrieben werden*)
ELSE
	Achs_State.PEH:=FALSE;
END_IF


KV_ANTEIL:=LIMIT( -KV2_LIMIT, (Achs_State.Schleppabst*KV2),KV2_LIMIT);

IF SET_P_T THEN
	D_Anteil:=0;
ELSE
	D_Anteil:=LREAL_TO_REAL((Achs_State.Vel_Ist-IV_RB.VEL_IST_LAST)/T_ZYKL*KD2);
END_IF

IF Antrieb_INVERS THEN
	Achs_to_DriveAdapter.motorSpeed:= LREAL_TO_REAL(-(Achs_State.Vel_Ist+KV_ANTEIL+D_Anteil) / mm_pro_MotUmdr*60);
	Achs_to_DriveAdapter.SA_MotUmdr:=LREAL_TO_REAL(-Achs_State.Schleppabst/mm_pro_MotUmdr);
ELSE
	Achs_to_DriveAdapter.motorSpeed:= LREAL_TO_REAL((Achs_State.Vel_Ist+KV_ANTEIL+D_Anteil) / mm_pro_MotUmdr*60);
	Achs_to_DriveAdapter.SA_MotUmdr:=LREAL_TO_REAL(Achs_State.Schleppabst/mm_pro_MotUmdr);
END_IF
END_ACTION

END_FUNCTION_BLOCK

// POUs/Nockenachsen/Nock_Incr_S_Achs
FUNCTION_BLOCK Nock_Incr_S_Achs
(* Invers Zählen wird durch Vertauschen von IN_A und IN_B erreicht; Achse Zählt vorwärts wenn die Signale von A nach B wandern, andernfalls rückwärts
Es wird Stillstand Überwacht für:	- Mechanische Blockade (keine Incremente beim vorfahren / keine Decremente beim zurückfahren für 2*T_pro_INC)
								- Ausfall der Spur A für 4*T_pro_INC
								- Ausfall der Spur B für 4*T_pro_INC
-T_pro INC sollte genau eingegeben werden, eventuell messen (TRACEaufzeichnung)
-S_STOP kann ermittelt werden, indem genau auf eine A-oderB-Spur-Flanke positioniert wird (z.B. auf REFPOS). 
Achtung: REFPOS ändert ONLINE die Istposition, muss deshalb konstant bleiben
27.04.2004
*)

VAR_INPUT
	DAT_FROM_PLC:TES_ACHSE_OUT;
	EREF: BOOL;
	IN_A: BOOL;(* Eingang Encoderspur A*)
	IN_B: BOOL;(* Eingang Encoderspur B*)
	IBW: LREAL; (*Istbewertung: mm/INREMENT *)
	T_pro_INC: LREAL; (* Zeitliche Abstand zwischen 2 Incrementen, dient zur WegIntrpolation*)
	S_STOP: REAL; (*Bremsweg Abschaltzeitpunkt bis zum Stillstand*)
	WAITTIME_INV: REAL; (* Wartezeit für Richtungsumkehr, dient zur schonung der Schütz und der Mechanik*)
	T_ZYKL: REAL;
	REFVEL1: INT;
	REFVEL2: INT;
END_VAR
VAR_OUTPUT
	DAT_TO_PLC:TES_ACHSE_IN;
	VOR_OUT: BOOL;
	ZUR_OUT: BOOL;
END_VAR
VAR
	V_SOLL:REAL;
	SYNC: BOOL;
	REFSTATUS: INT;
	IN_A_LAST: BOOL;
	IN_B_LAST: BOOL;
	INCR: BOOL;
	DECR: BOOL;
	IstPos: LREAL;
	IstIncr: DINT;
	T_seit_Letzt_EncFl: LREAL;
	PEH: BOOL;
	Zieldiff_Pos: LREAL;
	Start_Pos_LAST: BOOL;
	TIME_ZUR: REAL;
	TIME_VOR: REAL;
	T_STILLST: REAL;
	T_STILLST_A: REAL;
	T_STILLST_B: REAL;
END_VAR

